C03652=1137.389,195.650,-63.085,-178.221,7.484,148.898
C03653=1137.385,195.899,-63.109,-178.219,7.486,148.898
C03654=1137.380,196.148,-63.132,-178.216,7.489,148.898
C03655=1137.375,196.397,-63.157,-178.213,7.491,148.898
C03656=1137.371,196.646,-63.181,-178.210,7.493,148.898
C03657=1137.366,196.895,-63.204,-178.207,7.496,148.897
C03658=1137.362,197.143,-63.229,-178.204,7.499,148.897
C03659=1137.357,197.392,-63.254,-178.202,7.501,148.897
C03660=1137.353,197.641,-63.278,-178.199,7.504,148.897
C03661=1137.348,197.890,-63.301,-178.196,7.506,148.896
C03662=1137.343,198.138,-63.325,-178.193,7.508,148.896
C03663=1137.338,198.387,-63.350,-178.191,7.511,148.896
C03664=1137.335,198.636,-63.374,-178.187,7.514,148.896
C03665=1137.330,198.885,-63.398,-178.184,7.517,148.896
C03666=1137.325,199.134,-63.422,-178.182,7.518,148.895
C03667=1137.320,199.382,-63.446,-178.179,7.521,148.895
C03668=1137.317,199.631,-63.471,-178.176,7.524,148.895
C03669=1137.311,199.880,-63.495,-178.173,7.526,148.895
C03670=1137.307,200.129,-63.519,-178.171,7.529,148.895
C03671=1137.303,200.377,-63.544,-178.167,7.531,148.894
C03672=1137.298,200.627,-63.568,-178.165,7.533,148.894
C03673=1137.293,200.875,-63.592,-178.162,7.536,148.894
C03674=1137.289,201.124,-63.616,-178.159,7.539,148.894
C03675=1137.284,201.373,-63.641,-178.156,7.542,148.894
C03676=1137.280,201.622,-63.665,-178.154,7.544,148.894
C03677=1137.275,201.870,-63.690,-178.151,7.546,148.893
C03678=1137.271,202.119,-63.714,-178.148,7.549,148.893
C03679=1137.267,202.368,-63.738,-178.145,7.551,148.893
C03680=1137.262,202.617,-63.763,-178.142,7.554,148.893
C03681=1137.257,202.865,-63.787,-178.140,7.557,148.893
C03682=1137.253,203.115,-63.812,-178.136,7.559,148.892
C03683=1137.248,203.363,-63.836,-178.134,7.561,148.892
C03684=1137.243,203.612,-63.861,-178.131,7.564,148.892
C03685=1137.239,203.861,-63.885,-178.128,7.567,148.892
C03686=1137.234,204.110,-63.910,-178.125,7.570,148.892
C03687=1137.230,204.358,-63.934,-178.123,7.572,148.891
C03688=1137.226,204.607,-63.960,-178.120,7.574,148.891
C03689=1137.221,204.855,-63.984,-178.117,7.577,148.891
C03690=1137.216,205.104,-64.009,-178.114,7.580,148.891
C03691=1137.212,205.353,-64.033,-178.111,7.582,148.891
C03692=1137.207,205.602,-64.058,-178.109,7.585,148.890
C03693=1137.203,205.850,-64.082,-178.106,7.588,148.890
C03694=1137.198,206.100,-64.107,-178.102,7.590,148.890
C03695=1137.194,206.347,-64.132,-178.100,7.592,148.890
C03696=1137.189,206.596,-64.156,-178.097,7.595,148.890
C03697=1137.185,206.845,-64.181,-178.094,7.598,148.890
C03698=1137.180,207.094,-64.205,-178.091,7.601,148.889
C03699=1137.176,207.343,-64.230,-178.089,7.603,148.889
C03700=1137.171,207.591,-64.255,-178.086,7.605,148.889
C03701=1137.166,207.840,-64.280,-178.083,7.608,148.889
C03702=1137.162,208.089,-64.305,-178.080,7.611,148.889
C03703=1137.158,208.337,-64.330,-178.078,7.613,148.889
C03704=1137.153,208.586,-64.355,-178.075,7.616,148.888
C03705=1137.148,208.835,-64.379,-178.072,7.619,148.888
C03706=1137.144,209.106,-64.406,-178.069,7.622,148.888
C03707=1137.138,209.376,-64.433,-178.066,7.624,148.888
C03708=1137.134,209.647,-64.460,-178.063,7.627,148.888
C03709=1137.129,209.918,-64.487,-178.060,7.630,148.887
C03710=1137.124,210.166,-64.513,-178.057,7.632,148.887
C03711=1137.120,210.416,-64.538,-178.054,7.635,148.887
C03712=1137.115,210.664,-64.563,-178.051,7.638,148.887
C03713=1137.111,210.912,-64.587,-178.048,7.641,148.887
C03714=1137.106,211.161,-64.612,-178.046,7.643,148.887
C03715=1137.101,211.410,-64.638,-178.043,7.646,148.886
C03716=1137.097,211.659,-64.663,-178.040,7.649,148.886
C03717=1137.093,211.907,-64.687,-178.037,7.651,148.886
C03718=1137.088,212.156,-64.712,-178.034,7.654,148.886
C03719=1137.083,212.404,-64.738,-178.032,7.656,148.886
C03720=1137.079,212.654,-64.763,-178.029,7.659,148.886
C03721=1137.075,212.902,-64.788,-178.026,7.662,148.885
C03722=1137.070,213.151,-64.813,-178.023,7.665,148.885
C03723=1137.066,213.400,-64.838,-178.020,7.668,148.885
C03724=1137.061,213.648,-64.864,-178.017,7.670,148.885
C03725=1137.057,213.897,-64.889,-178.015,7.672,148.885
C03726=1137.052,214.145,-64.914,-178.012,7.675,148.885
C03727=1137.048,214.394,-64.939,-178.009,7.678,148.885
C03728=1137.043,214.643,-64.964,-178.006,7.681,148.884
C03729=1137.039,214.891,-64.990,-178.003,7.683,148.884
C03730=1137.034,215.141,-65.015,-178.001,7.686,148.884
C03731=1137.030,215.389,-65.040,-177.998,7.688,148.884
C03732=1137.025,215.638,-65.066,-177.995,7.691,148.884
C03733=1137.020,215.886,-65.091,-177.992,7.694,148.884
C03734=1137.017,216.135,-65.116,-177.989,7.697,148.883
C03735=1137.012,216.383,-65.141,-177.986,7.700,148.883
C03736=1137.008,216.632,-65.167,-177.984,7.702,148.883
C03737=1137.003,216.881,-65.192,-177.981,7.705,148.883
C03738=1136.998,217.129,-65.217,-177.978,7.707,148.883
C03739=1136.994,217.378,-65.243,-177.975,7.710,148.883
C03740=1136.990,217.627,-65.269,-177.972,7.713,148.883
C03741=1136.985,217.876,-65.294,-177.969,7.716,148.882
C03742=1136.981,218.125,-65.319,-177.967,7.719,148.882
C03743=1136.976,218.373,-65.345,-177.964,7.721,148.882
C03744=1136.971,218.621,-65.370,-177.961,7.723,148.882
C03745=1136.967,218.870,-65.396,-177.958,7.726,148.882
C03746=1136.963,219.119,-65.422,-177.956,7.729,148.882
C03747=1136.958,219.367,-65.447,-177.953,7.732,148.882
C03748=1136.954,219.617,-65.472,-177.950,7.735,148.882
C03749=1136.949,219.865,-65.498,-177.947,7.738,148.881
C03750=1136.945,220.113,-65.523,-177.944,7.740,148.881
C03751=1136.940,220.362,-65.549,-177.942,7.743,148.881
C03752=1136.936,220.611,-65.575,-177.939,7.746,148.881
C03753=1136.931,220.859,-65.600,-177.936,7.748,148.881
C03754=1136.927,221.108,-65.626,-177.933,7.751,148.881
C03755=1136.923,221.357,-65.652,-177.930,7.754,148.880
C03756=1136.917,221.605,-65.678,-177.927,7.757,148.880
C03757=1136.913,221.854,-65.704,-177.924,7.760,148.880
C03758=1136.909,222.103,-65.729,-177.922,7.762,148.880
C03759=1136.905,222.352,-65.755,-177.919,7.765,148.880
C03760=1136.900,222.600,-65.780,-177.917,7.768,148.880
C03761=1136.896,222.849,-65.806,-177.913,7.770,148.880
C03762=1136.891,223.097,-65.832,-177.910,7.773,148.880
C03763=1136.887,223.346,-65.858,-177.908,7.776,148.879
C03764=1136.882,223.594,-65.884,-177.905,7.779,148.879
C03765=1136.878,223.843,-65.910,-177.902,7.782,148.879
C03766=1136.873,224.092,-65.936,-177.900,7.784,148.879
C03767=1136.869,224.340,-65.962,-177.897,7.787,148.879
C03768=1136.864,224.588,-65.987,-177.894,7.790,148.879
C03769=1136.859,224.838,-66.013,-177.891,7.792,148.879
C03770=1136.855,225.086,-66.039,-177.888,7.795,148.879
C03771=1136.851,225.335,-66.066,-177.885,7.798,148.878
C03772=1136.847,225.583,-66.091,-177.882,7.801,148.878
C03773=1136.842,225.832,-66.117,-177.880,7.804,148.878
C03774=1136.837,226.081,-66.143,-177.877,7.807,148.878
C03775=1136.833,226.329,-66.170,-177.874,7.810,148.878
C03776=1136.829,226.578,-66.195,-177.871,7.813,148.878
C03777=1136.824,226.827,-66.222,-177.869,7.815,148.878
C03778=1136.820,227.076,-66.247,-177.866,7.817,148.878
C03779=1136.815,227.323,-66.274,-177.863,7.820,148.877
C03780=1136.810,227.572,-66.300,-177.860,7.823,148.877
C03781=1136.806,227.821,-66.326,-177.857,7.826,148.877
C03782=1136.802,228.069,-66.352,-177.855,7.829,148.877
C03783=1136.798,228.318,-66.378,-177.852,7.832,148.877
C03784=1136.793,228.567,-66.404,-177.849,7.835,148.877
C03785=1136.789,228.815,-66.431,-177.846,7.838,148.877
C03786=1136.784,229.064,-66.457,-177.843,7.840,148.877
C03787=1136.780,229.312,-66.483,-177.841,7.843,148.877
C03788=1136.776,229.561,-66.509,-177.838,7.846,148.877
C03789=1136.771,229.809,-66.536,-177.835,7.849,148.877
C03790=1136.767,230.058,-66.562,-177.832,7.851,148.876
C03791=1136.762,230.307,-66.587,-177.829,7.854,148.876
C03792=1136.758,230.555,-66.614,-177.827,7.857,148.876
C03793=1136.754,230.804,-66.640,-177.824,7.860,148.876
C03794=1136.749,231.052,-66.667,-177.821,7.863,148.876
C03795=1136.745,231.301,-66.694,-177.818,7.865,148.876
C03796=1136.740,231.550,-66.720,-177.815,7.868,148.876
C03797=1136.736,231.798,-66.747,-177.813,7.871,148.876
C03798=1136.731,232.046,-66.773,-177.810,7.874,148.876
C03799=1136.727,232.295,-66.799,-177.807,7.877,148.875
C03800=1136.722,232.544,-66.825,-177.804,7.880,148.875
C03801=1136.718,232.792,-66.852,-177.801,7.883,148.875
C03802=1136.713,233.040,-66.879,-177.799,7.886,148.875
C03803=1136.709,233.289,-66.905,-177.796,7.889,148.875
C03804=1136.704,233.538,-66.932,-177.793,7.892,148.875
C03805=1136.700,233.786,-66.957,-177.790,7.895,148.875
C03806=1136.695,234.035,-66.985,-177.787,7.897,148.875
C03807=1136.691,234.283,-67.011,-177.785,7.900,148.875
C03808=1136.687,234.532,-67.038,-177.782,7.903,148.875
C03809=1136.682,234.780,-67.064,-177.779,7.906,148.875
C03810=1136.678,235.053,-67.094,-177.776,7.909,148.874
C03811=1136.673,235.324,-67.123,-177.773,7.912,148.874
C03812=1136.667,235.597,-67.151,-177.769,7.915,148.874
C03813=1136.664,235.869,-67.181,-177.767,7.918,148.874
C03814=1136.659,236.117,-67.208,-177.764,7.921,148.874
C03815=1136.654,236.366,-67.235,-177.761,7.924,148.874
C03816=1136.650,236.614,-67.261,-177.758,7.927,148.874
C03817=1136.645,236.863,-67.288,-177.755,7.930,148.874
C03818=1136.641,237.111,-67.315,-177.753,7.933,148.874
C03819=1136.637,237.360,-67.341,-177.750,7.936,148.874
C03820=1136.632,237.608,-67.368,-177.747,7.939,148.874
C03821=1136.628,237.857,-67.395,-177.744,7.942,148.873
C03822=1136.624,238.105,-67.422,-177.741,7.944,148.873
C03823=1136.619,238.353,-67.449,-177.739,7.947,148.873
C03824=1136.614,238.602,-67.476,-177.736,7.950,148.873
C03825=1136.610,238.851,-67.502,-177.733,7.953,148.873
C03826=1136.606,239.100,-67.529,-177.730,7.956,148.873
C03827=1136.601,239.348,-67.556,-177.727,7.959,148.873
C03828=1136.597,239.597,-67.583,-177.725,7.962,148.873
C03829=1136.593,239.845,-67.610,-177.722,7.965,148.873
C03830=1136.588,240.093,-67.637,-177.719,7.968,148.873
C03831=1136.583,240.342,-67.664,-177.716,7.971,148.873
C03832=1136.579,240.590,-67.691,-177.713,7.974,148.873
C03833=1136.575,240.839,-67.717,-177.711,7.976,148.872
C03834=1136.571,241.088,-67.745,-177.708,7.979,148.872
C03835=1136.567,241.336,-67.772,-177.705,7.982,148.872
C03836=1136.562,241.584,-67.799,-177.702,7.985,148.872
C03837=1136.557,241.833,-67.827,-177.699,7.988,148.872
C03838=1136.553,242.081,-67.853,-177.697,7.991,148.872
C03839=1136.549,242.329,-67.880,-177.694,7.994,148.872
C03840=1136.545,242.578,-67.907,-177.691,7.997,148.872
C03841=1136.540,242.827,-67.935,-177.689,8.000,148.872
C03842=1136.535,243.075,-67.962,-177.686,8.003,148.872
C03843=1136.531,243.323,-67.989,-177.683,8.006,148.872
C03844=1136.527,243.572,-68.016,-177.680,8.009,148.872
C03845=1136.523,243.821,-68.043,-177.677,8.012,148.872
C03846=1136.518,244.069,-68.070,-177.675,8.015,148.872
C03847=1136.514,244.317,-68.098,-177.672,8.018,148.872
C03848=1136.509,244.566,-68.125,-177.669,8.020,148.871
C03849=1136.505,244.814,-68.152,-177.666,8.023,148.871
C03850=1136.501,245.063,-68.180,-177.663,8.026,148.871
C03851=1136.496,245.311,-68.207,-177.661,8.029,148.871
C03852=1136.492,245.560,-68.235,-177.658,8.032,148.871
C03853=1136.487,245.808,-68.262,-177.654,8.036,148.871
C03854=1136.483,246.057,-68.290,-177.652,8.039,148.871
C03855=1136.478,246.305,-68.317,-177.649,8.042,148.871
C03856=1136.474,246.554,-68.344,-177.646,8.045,148.871
C03857=1136.470,246.802,-68.372,-177.644,8.048,148.871
C03858=1136.465,247.051,-68.399,-177.641,8.051,148.871
C03859=1136.461,247.299,-68.426,-177.638,8.054,148.871
C03860=1136.456,247.547,-68.454,-177.635,8.057,148.871
C03861=1136.452,247.796,-68.481,-177.632,8.059,148.871
C03862=1136.448,248.044,-68.509,-177.630,8.062,148.871
C03863=1136.443,248.293,-68.536,-177.627,8.065,148.871
C03864=1136.440,248.541,-68.564,-177.624,8.068,148.871
C03865=1136.435,248.790,-68.591,-177.622,8.071,148.871
C03866=1136.431,249.038,-68.619,-177.619,8.074,148.871
C03867=1136.427,249.287,-68.647,-177.616,8.077,148.870
C03868=1136.422,249.535,-68.674,-177.613,8.080,148.870
C03869=1136.418,249.783,-68.701,-177.611,8.083,148.870
C03870=1136.414,250.032,-68.730,-177.607,8.087,148.870
C03871=1136.408,250.281,-68.757,-177.604,8.090,148.870
C03872=1136.404,250.529,-68.785,-177.602,8.093,148.870
C03873=1136.400,250.778,-68.812,-177.599,8.096,148.870
C03874=1136.396,251.026,-68.840,-177.596,8.099,148.870
C03875=1136.391,251.273,-68.868,-177.594,8.102,148.870
C03876=1136.387,251.523,-68.895,-177.591,8.105,148.870
C03877=1136.383,251.771,-68.923,-177.588,8.108,148.870
C03878=1136.378,252.019,-68.952,-177.585,8.110,148.870
C03879=1136.374,252.268,-68.979,-177.582,8.113,148.870
C03880=1136.369,252.516,-69.007,-177.580,8.116,148.870
C03881=1136.366,252.764,-69.035,-177.577,8.120,148.870
C03882=1136.361,253.013,-69.062,-177.574,8.123,148.870
C03883=1136.356,253.262,-69.091,-177.571,8.126,148.870
C03884=1136.352,253.510,-69.118,-177.568,8.129,148.870
C03885=1136.348,253.758,-69.146,-177.565,8.132,148.870
C03886=1136.344,254.007,-69.174,-177.563,8.135,148.870
C03887=1136.339,254.255,-69.202,-177.560,8.138,148.870
C03888=1136.335,254.503,-69.230,-177.557,8.141,148.870
C03889=1136.331,254.751,-69.258,-177.555,8.144,148.870
C03890=1136.327,255.000,-69.286,-177.552,8.147,148.870
C03891=1136.322,255.248,-69.314,-177.549,8.150,148.869
C03892=1136.318,255.497,-69.342,-177.546,8.154,148.869
C03893=1136.313,255.745,-69.370,-177.543,8.157,148.870
C03894=1136.309,255.994,-69.398,-177.541,8.160,148.870
C03895=1136.304,256.242,-69.426,-177.538,8.163,148.869
C03896=1136.301,256.491,-69.454,-177.535,8.166,148.869
C03897=1136.296,256.739,-69.483,-177.532,8.168,148.869
C03898=1136.292,256.987,-69.511,-177.530,8.172,148.869
C03899=1136.287,257.235,-69.539,-177.527,8.175,148.869
C03900=1136.283,257.484,-69.567,-177.524,8.178,148.869
C03901=1136.279,257.732,-69.595,-177.521,8.181,148.869
C03902=1136.274,257.981,-69.624,-177.518,8.184,148.869
C03903=1136.270,258.229,-69.652,-177.515,8.187,148.869
C03904=1136.266,258.477,-69.680,-177.513,8.190,148.869
C03905=1136.261,258.725,-69.708,-177.510,8.193,148.869
C03906=1136.257,258.974,-69.736,-177.507,8.196,148.869
C03907=1136.252,259.222,-69.765,-177.504,8.199,148.869
C03908=1136.248,259.471,-69.793,-177.502,8.203,148.869
C03909=1136.243,259.719,-69.821,-177.499,8.206,148.869
C03910=1136.240,259.968,-69.849,-177.496,8.209,148.869
C03911=1136.235,260.216,-69.878,-177.493,8.212,148.869
C03912=1136.231,260.464,-69.906,-177.490,8.215,148.869
C03913=1136.227,260.713,-69.935,-177.488,8.218,148.869
C03914=1136.222,260.986,-69.966,-177.485,8.222,148.869
C03915=1136.216,261.260,-69.997,-177.482,8.225,148.869
C03916=1136.212,261.534,-70.028,-177.478,8.228,148.869
C03917=1136.207,261.807,-70.060,-177.475,8.232,148.869
C03918=1136.204,262.055,-70.088,-177.473,8.235,148.869
C03919=1136.199,262.304,-70.117,-177.470,8.238,148.869
C03920=1136.195,262.552,-70.145,-177.467,8.241,148.869
C03921=1136.191,262.800,-70.174,-177.464,8.244,148.869
C03922=1136.185,263.048,-70.203,-177.462,8.247,148.869
C03923=1136.182,263.297,-70.231,-177.459,8.251,148.869
C03924=1136.178,263.545,-70.260,-177.456,8.254,148.869
C03925=1136.173,263.793,-70.288,-177.453,8.257,148.869
C03926=1136.169,264.042,-70.317,-177.451,8.260,148.869
C03927=1136.165,264.290,-70.346,-177.448,8.263,148.869
C03928=1136.160,264.538,-70.374,-177.445,8.266,148.869
C03929=1136.156,264.787,-70.403,-177.442,8.270,148.869
C03930=1136.151,265.035,-70.432,-177.439,8.273,148.869
C03931=1136.147,265.283,-70.460,-177.437,8.276,148.869
C03932=1136.143,265.531,-70.490,-177.434,8.279,148.869
C03933=1136.138,265.780,-70.518,-177.431,8.282,148.869
C03934=1136.134,266.028,-70.546,-177.429,8.285,148.869
C03935=1136.130,266.277,-70.575,-177.425,8.289,148.869
C03936=1136.125,266.525,-70.604,-177.422,8.292,148.869
C03937=1136.121,266.774,-70.634,-177.420,8.295,148.869
C03938=1136.117,267.022,-70.661,-177.417,8.298,148.869
C03939=1136.113,267.270,-70.691,-177.414,8.301,148.869
C03940=1136.108,267.519,-70.720,-177.412,8.305,148.869
C03941=1136.103,267.766,-70.749,-177.409,8.308,148.869
C03942=1136.100,268.015,-70.777,-177.406,8.311,148.869
C03943=1136.096,268.263,-70.806,-177.404,8.314,148.869
C03944=1136.091,268.511,-70.836,-177.401,8.317,148.869
C03945=1136.086,268.760,-70.864,-177.397,8.321,148.869
C03946=1136.083,269.008,-70.893,-177.395,8.324,148.869
C03947=1136.079,269.256,-70.922,-177.392,8.327,148.869
C03948=1136.074,269.505,-70.951,-177.389,8.330,148.869
C03949=1136.070,269.753,-70.981,-177.387,8.333,148.869
C03950=1136.065,270.001,-71.009,-177.384,8.337,148.869
C03951=1136.061,270.249,-71.038,-177.381,8.340,148.869
C03952=1136.057,270.497,-71.067,-177.378,8.342,148.869
C03953=1136.053,270.746,-71.097,-177.376,8.346,148.869
C03954=1136.049,270.995,-71.126,-177.373,8.349,148.869
C03955=1136.044,271.242,-71.155,-177.370,8.353,148.869
C03956=1136.040,271.490,-71.184,-177.367,8.356,148.869
C03957=1136.035,271.739,-71.214,-177.365,8.359,148.869
C03958=1136.031,271.987,-71.242,-177.362,8.362,148.869
C03959=1136.027,272.236,-71.272,-177.359,8.365,148.869
C03960=1136.023,272.484,-71.301,-177.356,8.368,148.869
C03961=1136.019,272.731,-71.330,-177.354,8.372,148.870
C03962=1136.014,272.980,-71.359,-177.351,8.375,148.870
C03963=1136.010,273.228,-71.389,-177.348,8.378,148.869
C03964=1136.006,273.477,-71.417,-177.345,8.382,148.870
C03965=1136.002,273.725,-71.447,-177.342,8.385,148.870
C03966=1135.997,273.973,-71.476,-177.340,8.388,148.870
C03967=1135.993,274.222,-71.506,-177.337,8.391,148.870
C03968=1135.989,274.470,-71.535,-177.334,8.394,148.870
C03969=1135.985,274.718,-71.565,-177.331,8.398,148.870
C03970=1135.980,274.966,-71.594,-177.329,8.401,148.870
C03971=1135.976,275.214,-71.623,-177.326,8.404,148.870
C03972=1135.972,275.462,-71.653,-177.323,8.408,148.870
C03973=1135.967,275.710,-71.682,-177.320,8.410,148.870
C03974=1135.963,275.959,-71.711,-177.318,8.414,148.870
C03975=1135.959,276.207,-71.741,-177.315,8.417,148.870
C03976=1135.954,276.456,-71.771,-177.312,8.421,148.870
C03977=1135.950,276.704,-71.800,-177.309,8.424,148.870
C03978=1135.946,276.952,-71.830,-177.306,8.427,148.870
C03979=1135.942,277.200,-71.859,-177.304,8.430,148.870
C03980=1135.937,277.449,-71.889,-177.301,8.434,148.870
C03981=1135.934,277.696,-71.919,-177.298,8.437,148.870
C03982=1135.929,277.945,-71.948,-177.296,8.440,148.870
C03983=1135.925,278.193,-71.978,-177.293,8.443,148.870
C03984=1135.921,278.441,-72.007,-177.290,8.447,148.870
C03985=1135.917,278.689,-72.037,-177.287,8.450,148.870
C03986=1135.912,278.938,-72.067,-177.285,8.453,148.871
C03987=1135.908,279.186,-72.097,-177.282,8.456,148.870
C03988=1135.904,279.434,-72.126,-177.279,8.460,148.871
C03989=1135.900,279.682,-72.156,-177.276,8.463,148.871
C03990=1135.896,279.930,-72.185,-177.274,8.466,148.871
C03991=1135.891,280.179,-72.215,-177.270,8.470,148.871
C03992=1135.887,280.427,-72.246,-177.268,8.473,148.871
C03993=1135.883,280.675,-72.275,-177.265,8.476,148.871
C03994=1135.878,280.923,-72.304,-177.263,8.479,148.871
C03995=1135.874,281.171,-72.335,-177.260,8.483,148.871
C03996=1135.870,281.419,-72.365,-177.257,8.486,148.871
C03997=1135.865,281.668,-72.394,-177.254,8.489,148.871
C03998=1135.862,281.915,-72.424,-177.251,8.493,148.871
C03999=1135.857,282.164,-72.454,-177.249,8.496,148.871
C04000=1135.852,282.412,-72.484,-177.246,8.499,148.871
C04001=1135.849,282.660,-72.514,-177.244,8.502,148.871
C04002=1135.844,282.908,-72.544,-177.240,8.506,148.871
C04003=1135.840,283.156,-72.574,-177.238,8.509,148.872
C04004=1135.836,283.405,-72.604,-177.235,8.512,148.871
C04005=1135.832,283.653,-72.635,-177.232,8.516,148.872
C04006=1135.825,284.060,-72.683,-177.228,8.522,148.872
C04007=1135.804,285.282,-72.833,-178.121,10.280,149.550
C04008=1135.800,285.531,-72.864,-178.118,10.283,149.550
C04009=1135.796,285.779,-72.894,-178.115,10.285,149.550
C04010=1135.791,286.027,-72.925,-178.112,10.288,149.550
C04011=1135.786,286.275,-72.955,-178.109,10.290,149.550
C04012=1135.783,286.524,-72.986,-178.106,10.293,149.549
C04013=1135.779,286.772,-73.017,-178.103,10.296,149.549
C04014=1135.775,287.019,-73.047,-178.100,10.298,149.549
C04015=1135.771,287.268,-73.078,-178.096,10.301,149.549
C04016=1135.766,287.516,-73.109,-178.093,10.304,149.549
C04017=1135.762,287.763,-73.139,-178.091,10.305,149.548
C04018=1135.758,288.012,-73.170,-178.088,10.308,149.548
C04019=1135.754,288.260,-73.201,-178.084,10.310,149.548
C04020=1135.750,288.508,-73.231,-178.081,10.313,149.548
C04021=1135.746,288.756,-73.262,-178.078,10.316,149.548
C04022=1135.741,289.004,-73.293,-178.075,10.318,149.548
C04023=1135.736,289.252,-73.324,-178.072,10.321,149.547
C04024=1135.733,289.501,-73.354,-178.069,10.324,149.547
C04025=1135.729,289.748,-73.386,-178.066,10.326,149.547
C04026=1135.724,289.996,-73.416,-178.063,10.329,149.547
C04027=1135.720,290.245,-73.448,-178.060,10.331,149.547
C04028=1135.716,290.492,-73.478,-178.056,10.334,149.546
C04029=1135.712,290.740,-73.508,-178.054,10.336,149.546
C04030=1135.708,290.989,-73.540,-178.051,10.338,149.546
C04031=1135.703,291.236,-73.571,-178.048,10.341,149.546
C04032=1135.700,291.485,-73.602,-178.044,10.343,149.546
C04033=1135.696,291.732,-73.632,-178.041,10.346,149.546
C04034=1135.691,291.980,-73.663,-178.038,10.349,149.545
C04035=1135.687,292.229,-73.694,-178.035,10.351,149.545
C04036=1135.683,292.476,-73.726,-178.032,10.354,149.545
C04037=1135.679,292.725,-73.757,-178.029,10.357,149.545
C04038=1135.675,292.973,-73.787,-178.026,10.359,149.545
C04039=1135.671,293.221,-73.819,-178.023,10.362,149.544
C04040=1135.667,293.452,-73.847,-178.020,10.364,149.544
C04041=1135.663,293.683,-73.877,-178.017,10.366,149.544
C04042=1135.659,293.914,-73.905,-178.014,10.369,149.544
C04043=1135.656,294.145,-73.935,-178.012,10.371,149.544
C04044=1135.651,294.377,-73.964,-178.008,10.373,149.544
C04045=1135.647,294.607,-73.993,-178.005,10.376,149.544
C04046=1135.643,294.839,-74.021,-178.003,10.378,149.543
C04047=1135.639,295.070,-74.051,-178.000,10.381,149.543
C04048=1135.636,295.318,-74.083,-177.996,10.383,149.543
C04049=1135.631,295.566,-74.113,-177.994,10.386,149.543
C04050=1135.627,295.814,-74.144,-177.991,10.389,149.543
C04051=1135.623,296.062,-74.176,-177.987,10.391,149.542
C04052=1135.619,296.310,-74.207,-177.984,10.394,149.542
C04053=1135.614,296.558,-74.239,-177.981,10.396,149.542
C04054=1135.610,296.806,-74.270,-177.979,10.398,149.542
C04055=1135.606,297.054,-74.301,-177.975,10.401,149.542
C04056=1135.602,297.302,-74.332,-177.972,10.403,149.542
C04057=1135.598,297.550,-74.364,-177.969,10.406,149.541
C04058=1135.594,297.798,-74.396,-177.966,10.408,149.541
C04059=1135.590,298.046,-74.426,-177.963,10.411,149.541
C04060=1135.586,298.294,-74.458,-177.959,10.413,149.541
C04061=1135.581,298.542,-74.489,-177.957,10.416,149.541
C04062=1135.578,298.790,-74.521,-177.953,10.419,149.540
C04063=1135.573,299.037,-74.552,-177.950,10.421,149.540
C04064=1135.569,299.286,-74.583,-177.947,10.424,149.540
C04065=1135.565,299.533,-74.615,-177.944,10.427,149.540
C04066=1135.561,299.781,-74.647,-177.941,10.429,149.540
C04067=1135.557,300.030,-74.678,-177.938,10.432,149.540
C04068=1135.553,300.277,-74.709,-177.934,10.434,149.539
C04069=1135.549,300.525,-74.741,-177.931,10.437,149.539
C04070=1135.544,300.773,-74.773,-177.929,10.439,149.539
C04071=1135.540,301.021,-74.804,-177.926,10.441,149.539
C04072=1135.536,301.269,-74.836,-177.922,10.444,149.539
C04073=1135.532,301.517,-74.868,-177.920,10.447,149.538
C04074=1135.528,301.765,-74.900,-177.916,10.449,149.538
C04075=1135.524,302.013,-74.930,-177.913,10.452,149.538
C04076=1135.519,302.261,-74.963,-177.910,10.454,149.538
C04077=1135.516,302.509,-74.995,-177.907,10.457,149.538
C04078=1135.511,302.756,-75.026,-177.904,10.459,149.538
C04079=1135.508,303.004,-75.058,-177.900,10.462,149.537
C04080=1135.503,303.253,-75.090,-177.897,10.465,149.537
C04081=1135.499,303.501,-75.121,-177.894,10.467,149.537
C04082=1135.495,303.749,-75.153,-177.891,10.470,149.537
C04083=1135.491,303.997,-75.185,-177.888,10.472,149.537
C04084=1135.486,304.245,-75.217,-177.885,10.475,149.536
C04085=1135.482,304.493,-75.249,-177.882,10.477,149.536
C04086=1135.479,304.741,-75.281,-177.879,10.479,149.536
C04087=1135.474,304.988,-75.312,-177.876,10.482,149.536
C04088=1135.470,305.236,-75.345,-177.873,10.485,149.536
C04089=1135.466,305.484,-75.376,-177.870,10.487,149.536
C04090=1135.462,305.732,-75.408,-177.866,10.489,149.535
C04091=1135.457,305.980,-75.440,-177.863,10.492,149.535
C04092=1135.454,306.228,-75.472,-177.860,10.495,149.535
C04093=1135.449,306.475,-75.504,-177.857,10.497,149.535
C04094=1135.445,306.724,-75.536,-177.854,10.500,149.535
C04095=1135.441,306.972,-75.568,-177.851,10.503,149.534
C04096=1135.437,307.185,-75.596,-177.848,10.504,149.534
C04097=1135.434,307.398,-75.624,-177.845,10.507,149.534
C04098=1135.430,307.613,-75.651,-177.843,10.509,149.534
C04099=1135.427,307.826,-75.679,-177.840,10.511,149.534
C04100=1135.423,308.039,-75.707,-177.837,10.513,149.534
C04101=1135.420,308.253,-75.734,-177.835,10.515,149.534
C04102=1135.416,308.467,-75.762,-177.832,10.518,149.533
C04103=1135.414,308.681,-75.790,-177.829,10.520,149.533
C04104=1135.409,308.928,-75.822,-177.826,10.522,149.533
C04105=1135.405,309.176,-75.854,-177.823,10.525,149.533
C04106=1135.400,309.425,-75.886,-177.820,10.527,149.533
C04107=1135.397,309.673,-75.918,-177.816,10.530,149.532
C04108=1135.392,309.920,-75.951,-177.814,10.533,149.532
C04109=1135.388,310.168,-75.983,-177.810,10.535,149.532
C04110=1135.384,310.416,-76.015,-177.807,10.538,149.532
C04111=1135.380,310.663,-76.048,-177.804,10.540,149.532
C04112=1135.376,310.912,-76.080,-177.801,10.543,149.532
C04113=1135.372,311.160,-76.112,-177.798,10.546,149.531
C04114=1135.368,311.407,-76.145,-177.794,10.548,149.531
C04115=1135.364,311.655,-76.177,-177.791,10.551,149.531
C04116=1135.359,311.903,-76.209,-177.788,10.553,149.531
C04117=1135.356,312.151,-76.242,-177.785,10.556,149.531
C04118=1135.352,312.399,-76.274,-177.782,10.558,149.530
C04119=1135.348,312.646,-76.307,-177.779,10.560,149.530
C04120=1135.343,312.894,-76.339,-177.776,10.563,149.530
C04121=1135.339,313.142,-76.371,-177.773,10.565,149.530
C04122=1135.335,313.390,-76.404,-177.770,10.568,149.530
C04123=1135.331,313.638,-76.436,-177.767,10.570,149.529
C04124=1135.327,313.886,-76.469,-177.763,10.573,149.529
C04125=1135.323,314.134,-76.501,-177.760,10.576,149.529
C04126=1135.320,314.381,-76.534,-177.757,10.578,149.529
C04127=1135.315,314.630,-76.566,-177.754,10.581,149.529
C04128=1135.311,314.878,-76.599,-177.751,10.583,149.528
C04129=1135.307,315.126,-76.631,-177.747,10.586,149.528
C04130=1135.303,315.373,-76.664,-177.744,10.589,149.528
C04131=1135.298,315.620,-76.697,-177.741,10.591,149.528
C04132=1135.295,315.868,-76.729,-177.738,10.593,149.528
C04133=1135.291,316.116,-76.762,-177.735,10.596,149.528
C04134=1135.286,316.364,-76.794,-177.732,10.599,149.527
C04135=1135.283,316.612,-76.827,-177.729,10.601,149.527
C04136=1135.279,316.860,-76.860,-177.725,10.604,149.527
C04137=1135.274,317.108,-76.893,-177.722,10.606,149.527
C04138=1135.271,317.355,-76.925,-177.719,10.609,149.527
C04139=1135.267,317.603,-76.958,-177.716,10.611,149.526
C04140=1135.262,317.851,-76.992,-177.712,10.614,149.526
C04141=1135.258,318.099,-77.024,-177.710,10.616,149.526
C04142=1135.255,318.347,-77.057,-177.707,10.618,149.526
C04143=1135.250,318.594,-77.090,-177.703,10.621,149.526
C04144=1135.246,318.842,-77.123,-177.701,10.624,149.525
C04145=1135.242,319.090,-77.155,-177.697,10.626,149.525
C04146=1135.238,319.338,-77.188,-177.694,10.628,149.525
C04147=1135.234,319.586,-77.221,-177.691,10.631,149.525
C04148=1135.230,319.833,-77.254,-177.688,10.634,149.525
C04149=1135.226,320.081,-77.287,-177.684,10.636,149.524
C04150=1135.222,320.329,-77.320,-177.681,10.639,149.524
C04151=1135.217,320.577,-77.353,-177.678,10.641,149.524
C04152=1135.214,320.790,-77.382,-177.676,10.643,149.524
C04153=1135.211,321.004,-77.410,-177.672,10.646,149.524
C04154=1135.208,321.217,-77.438,-177.670,10.648,149.524
C04155=1135.204,321.430,-77.467,-177.667,10.650,149.523
C04156=1135.201,321.644,-77.495,-177.665,10.652,149.523
C04157=1135.197,321.858,-77.523,-177.662,10.655,149.523
C04158=1135.194,322.071,-77.552,-177.659,10.657,149.523
C04159=1135.190,322.285,-77.581,-177.657,10.659,149.523
C04160=1135.186,322.533,-77.614,-177.653,10.661,149.523
C04161=1135.182,322.781,-77.647,-177.650,10.663,149.522
C04162=1135.178,323.028,-77.680,-177.647,10.666,149.522
C04163=1135.174,323.276,-77.714,-177.644,10.669,149.522
C04164=1135.170,323.523,-77.746,-177.640,10.671,149.522
C04165=1135.166,323.771,-77.779,-177.637,10.674,149.522
C04166=1135.162,324.019,-77.812,-177.634,10.676,149.521
C04167=1135.158,324.266,-77.846,-177.631,10.679,149.521
C04168=1135.155,324.514,-77.880,-177.628,10.682,149.521
C04169=1135.151,324.762,-77.913,-177.625,10.684,149.521
C04170=1135.146,325.010,-77.946,-177.621,10.686,149.521
C04171=1135.142,325.258,-77.979,-177.618,10.689,149.520
C04172=1135.138,325.505,-78.012,-177.615,10.692,149.520
C04173=1135.134,325.753,-78.046,-177.612,10.694,149.520
C04174=1135.130,326.000,-78.079,-177.608,10.697,149.520
C04175=1135.127,326.249,-78.113,-177.605,10.699,149.520
C04176=1135.123,326.496,-78.146,-177.602,10.702,149.520
C04177=1135.118,326.744,-78.180,-177.599,10.704,149.519
C04178=1135.113,326.992,-78.213,-177.596,10.707,149.519
C04179=1135.110,327.239,-78.247,-177.593,10.709,149.519
C04180=1135.106,327.487,-78.280,-177.589,10.712,149.519
C04181=1135.102,327.735,-78.314,-177.586,10.714,149.518
C04182=1135.098,327.982,-78.347,-177.583,10.717,149.518
C04183=1135.094,328.230,-78.381,-177.580,10.720,149.518
C04184=1135.090,328.478,-78.414,-177.576,10.722,149.518
C04185=1135.086,328.725,-78.448,-177.573,10.725,149.518
C04186=1135.082,328.974,-78.482,-177.570,10.727,149.518
C04187=1135.078,329.221,-78.515,-177.567,10.729,149.517
C04188=1135.074,329.469,-78.549,-177.564,10.731,149.517
C04189=1135.070,329.716,-78.582,-177.561,10.734,149.517
C04190=1135.066,329.965,-78.615,-177.558,10.737,149.517
C04191=1135.062,330.212,-78.649,-177.554,10.739,149.517
C04192=1135.057,330.460,-78.683,-177.551,10.741,149.516
C04193=1135.054,330.707,-78.717,-177.548,10.744,149.516
C04194=1135.050,330.955,-78.750,-177.545,10.747,149.516
C04195=1135.046,331.203,-78.784,-177.542,10.749,149.516
C04196=1135.041,331.451,-78.818,-177.538,10.752,149.516
C04197=1135.038,331.698,-78.852,-177.535,10.754,149.515
C04198=1135.034,331.946,-78.885,-177.532,10.757,149.515
C04199=1135.030,332.193,-78.919,-177.529,10.759,149.515
C04200=1135.025,332.441,-78.953,-177.525,10.762,149.515
C04201=1135.021,332.688,-78.987,-177.522,10.765,149.515
C04202=1135.018,332.936,-79.021,-177.519,10.767,149.514
C04203=1135.014,333.184,-79.054,-177.516,10.769,149.514
C04204=1135.009,333.431,-79.089,-177.512,10.772,149.514
C04205=1135.006,333.680,-79.122,-177.510,10.775,149.514
C04206=1135.002,333.927,-79.156,-177.506,10.777,149.514
C04207=1134.998,334.174,-79.191,-177.503,10.780,149.513
C04208=1134.995,334.388,-79.220,-177.501,10.782,149.513
C04209=1134.991,334.601,-79.249,-177.497,10.784,149.513
C04210=1134.987,334.815,-79.279,-177.495,10.786,149.513
C04211=1134.985,335.028,-79.308,-177.492,10.788,149.513
C04212=1134.981,335.241,-79.337,-177.489,10.790,149.513
C04213=1134.977,335.455,-79.367,-177.486,10.793,149.512
C04214=1134.974,335.668,-79.396,-177.483,10.795,149.512
C04215=1134.971,335.882,-79.425,-177.481,10.797,149.512
C04216=1134.966,336.129,-79.459,-177.478,10.799,149.512
C04217=1134.963,336.376,-79.493,-177.474,10.801,149.512
C04218=1134.959,336.624,-79.527,-177.472,10.804,149.512
C04219=1134.954,336.872,-79.561,-177.468,10.807,149.511
C04220=1134.951,337.120,-79.595,-177.465,10.809,149.511
C04221=1134.947,337.367,-79.630,-177.462,10.812,149.511
C04222=1134.943,337.614,-79.664,-177.458,10.814,149.511
C04223=1134.939,337.862,-79.699,-177.455,10.817,149.511
C04224=1134.935,338.109,-79.732,-177.452,10.819,149.510
C04225=1134.931,338.358,-79.767,-177.449,10.822,149.510
C04226=1134.927,338.605,-79.801,-177.445,10.824,149.510
C04227=1134.923,338.853,-79.835,-177.442,10.827,149.510
C04228=1134.919,339.101,-79.869,-177.439,10.829,149.510
C04229=1134.914,339.348,-79.904,-177.436,10.832,149.509
C04230=1134.911,339.596,-79.938,-177.433,10.834,149.509
C04231=1134.907,339.843,-79.972,-177.429,10.837,149.509
C04232=1134.903,340.091,-80.006,-177.426,10.839,149.509
C04233=1134.899,340.338,-80.041,-177.423,10.842,149.508
C04234=1134.895,340.587,-80.076,-177.420,10.844,149.508
C04235=1134.891,340.834,-80.110,-177.416,10.847,149.508
C04236=1134.887,341.081,-80.145,-177.413,10.849,149.508
C04237=1134.884,341.328,-80.179,-177.410,10.852,149.508
C04238=1134.880,341.576,-80.214,-177.406,10.854,149.507
C04239=1134.875,341.824,-80.248,-177.403,10.857,149.507
C04240=1134.872,342.072,-80.283,-177.400,10.860,149.507
C04241=1134.867,342.319,-80.317,-177.397,10.862,149.507
C04242=1134.863,342.567,-80.352,-177.394,10.864,149.507
C04243=1134.859,342.814,-80.386,-177.390,10.867,149.506
C04244=1134.856,343.062,-80.421,-177.387,10.869,149.506
C04245=1134.851,343.309,-80.456,-177.384,10.872,149.506
C04246=1134.848,343.557,-80.490,-177.381,10.875,149.506
C04247=1134.843,343.804,-80.524,-177.377,10.877,149.506
C04248=1134.839,344.053,-80.559,-177.374,10.880,149.505
C04249=1134.836,344.299,-80.594,-177.371,10.882,149.505
C04250=1134.832,344.547,-80.629,-177.367,10.884,149.505
C04251=1134.827,344.795,-80.663,-177.364,10.887,149.505
C04252=1134.824,345.042,-80.698,-177.361,10.889,149.504
C04253=1134.820,345.289,-80.733,-177.358,10.892,149.504
C04254=1134.816,345.537,-80.767,-177.355,10.895,149.504
C04255=1134.812,345.785,-80.803,-177.351,10.897,149.504
C04256=1134.808,346.032,-80.837,-177.348,10.899,149.504
C04257=1134.804,346.280,-80.872,-177.345,10.902,149.503
C04258=1134.800,346.527,-80.907,-177.341,10.904,149.503
C04259=1134.796,346.775,-80.942,-177.339,10.906,149.503
C04260=1134.792,347.023,-80.977,-177.335,10.909,149.503
C04261=1134.789,347.270,-81.011,-177.332,10.911,149.503
C04262=1134.785,347.518,-81.046,-177.329,10.914,149.502
C04263=1134.780,347.764,-81.081,-177.326,10.916,149.502
C04264=1134.777,347.978,-81.112,-177.322,10.919,149.502
C04265=1134.773,348.192,-81.142,-177.320,10.921,149.502
C04266=1134.771,348.405,-81.172,-177.317,10.923,149.502
C04267=1134.767,348.617,-81.202,-177.314,10.925,149.501
C04268=1134.763,348.831,-81.232,-177.311,10.928,149.501
C04269=1134.760,349.044,-81.262,-177.309,10.929,149.501
C04270=1134.757,349.257,-81.292,-177.306,10.931,149.501
C04271=1134.754,349.471,-81.323,-177.303,10.934,149.501
C04272=1134.749,349.718,-81.357,-177.299,10.936,149.500
C04273=1134.746,349.966,-81.393,-177.295,10.939,149.500
C04274=1134.742,350.213,-81.428,-177.292,10.942,149.500
C04275=1134.737,350.460,-81.463,-177.288,10.945,149.500
C04276=1134.734,350.708,-81.498,-177.284,10.947,149.499
C04277=1134.730,350.955,-81.534,-177.280,10.950,149.499
C04278=1134.726,351.203,-81.568,-177.277,10.953,149.499
C04279=1134.722,351.450,-81.604,-177.273,10.956,149.499
C04280=1134.719,351.698,-81.639,-177.269,10.958,149.498
C04281=1134.715,351.946,-81.674,-177.266,10.961,149.498
C04282=1134.711,352.193,-81.709,-177.262,10.963,149.498
C04283=1134.707,352.440,-81.744,-177.258,10.967,149.498
C04284=1134.703,352.688,-81.780,-177.255,10.969,149.497
C04285=1134.699,352.936,-81.815,-177.251,10.971,149.497
C04286=1134.694,353.183,-81.850,-177.247,10.974,149.497
C04287=1134.691,353.430,-81.886,-177.244,10.977,149.497
C04288=1134.687,353.678,-81.922,-177.240,10.979,149.496
C04289=1134.683,353.925,-81.957,-177.236,10.982,149.496
C04290=1134.679,354.172,-81.992,-177.233,10.985,149.496
C04291=1134.676,354.420,-82.028,-177.229,10.987,149.495
C04292=1134.672,354.668,-82.063,-177.225,10.990,149.495
C04293=1134.668,354.915,-82.098,-177.222,10.993,149.495
C04294=1134.664,355.163,-82.134,-177.218,10.995,149.494
C04295=1134.660,355.409,-82.169,-177.215,10.997,149.494
C04296=1134.656,355.657,-82.205,-177.211,11.000,149.494
C04297=1134.653,355.904,-82.240,-177.207,11.003,149.494
C04298=1134.648,356.152,-82.276,-177.204,11.005,149.493
C04299=1134.645,356.400,-82.312,-177.200,11.008,149.493
C04300=1134.641,356.647,-82.347,-177.196,11.011,149.493
C04301=1134.637,356.894,-82.382,-177.193,11.013,149.493
C04302=1134.633,357.142,-82.418,-177.189,11.015,149.492
C04303=1134.629,357.389,-82.454,-177.186,11.018,149.492
C04304=1134.625,357.636,-82.490,-177.182,11.020,149.492
C04305=1134.622,357.884,-82.526,-177.179,11.023,149.492
C04306=1134.618,358.131,-82.562,-177.175,11.026,149.491
C04307=1134.614,358.379,-82.597,-177.171,11.028,149.491
C04308=1134.610,358.627,-82.633,-177.168,11.030,149.491
C04309=1134.606,358.873,-82.668,-177.165,11.033,149.491
C04310=1134.602,359.121,-82.704,-177.162,11.035,149.490
C04311=1134.599,359.368,-82.740,-177.158,11.037,149.490
C04312=1134.594,359.616,-82.776,-177.155,11.040,149.490
C04313=1134.591,359.863,-82.812,-177.151,11.042,149.489
C04314=1134.587,360.111,-82.847,-177.148,11.044,149.489
C04315=1134.583,360.357,-82.884,-177.144,11.048,149.489
C04316=1134.579,360.605,-82.920,-177.140,11.050,149.489
C04317=1134.575,360.853,-82.955,-177.137,11.053,149.488
C04318=1134.572,361.100,-82.992,-177.133,11.055,149.488
C04319=1134.568,361.347,-83.028,-177.130,11.057,149.488
C04320=1134.564,361.561,-83.058,-177.127,11.059,149.488
C04321=1134.561,361.773,-83.090,-177.124,11.061,149.487
C04322=1134.558,361.987,-83.120,-177.122,11.063,149.487
C04323=1134.555,362.199,-83.151,-177.119,11.065,149.487
C04324=1134.552,362.413,-83.182,-177.116,11.068,149.487
C04325=1134.548,362.626,-83.214,-177.113,11.069,149.487
C04326=1134.544,362.839,-83.244,-177.110,11.072,149.486
C04327=1134.541,363.052,-83.276,-177.107,11.073,149.486
C04328=1134.538,363.299,-83.311,-177.104,11.076,149.486
C04329=1134.534,363.546,-83.348,-177.100,11.078,149.486
C04330=1134.530,363.794,-83.384,-177.097,11.080,149.485
C04331=1134.527,364.041,-83.420,-177.093,11.083,149.485
C04332=1134.522,364.288,-83.456,-177.090,11.085,149.485
C04333=1134.519,364.535,-83.492,-177.087,11.088,149.485
C04334=1134.514,364.783,-83.529,-177.084,11.090,149.484
C04335=1134.511,365.030,-83.565,-177.081,11.092,149.484
C04336=1134.507,365.277,-83.602,-177.078,11.095,149.484
C04337=1134.503,365.525,-83.637,-177.074,11.097,149.484
C04338=1134.499,365.772,-83.674,-177.071,11.099,149.483
C04339=1134.496,366.019,-83.710,-177.067,11.102,149.483
C04340=1134.491,366.267,-83.746,-177.064,11.104,149.483
C04341=1134.489,366.514,-83.783,-177.061,11.106,149.483
C04342=1134.484,366.762,-83.819,-177.058,11.108,149.482
C04343=1134.481,367.009,-83.855,-177.055,11.111,149.482
C04344=1134.477,367.256,-83.892,-177.051,11.113,149.482
C04345=1134.473,367.503,-83.928,-177.048,11.116,149.482
C04346=1134.469,367.751,-83.965,-177.045,11.117,149.482
C04347=1134.465,367.998,-84.002,-177.042,11.120,149.481
C04348=1134.461,368.245,-84.037,-177.039,11.122,149.481
C04349=1134.457,368.493,-84.074,-177.036,11.125,149.481
C04350=1134.454,368.739,-84.110,-177.033,11.126,149.481
C04351=1134.450,368.987,-84.147,-177.030,11.129,149.480
C04352=1134.446,369.235,-84.184,-177.026,11.131,149.480
C04353=1134.443,369.482,-84.220,-177.024,11.133,149.480
C04354=1134.439,369.729,-84.257,-177.020,11.136,149.480
C04355=1134.434,369.976,-84.294,-177.017,11.138,149.480
C04356=1134.431,370.223,-84.330,-177.014,11.141,149.479
C04357=1134.427,370.470,-84.367,-177.011,11.142,149.479
C04358=1134.423,370.718,-84.403,-177.008,11.145,149.479
C04359=1134.420,370.966,-84.440,-177.005,11.148,149.479
C04360=1134.416,371.213,-84.476,-177.002,11.149,149.479
C04361=1134.412,371.460,-84.513,-176.999,11.152,149.478
C04362=1134.408,371.707,-84.549,-176.996,11.154,149.478
C04363=1134.404,371.954,-84.586,-176.993,11.156,149.478
C04364=1134.400,372.202,-84.623,-176.990,11.158,149.478
C04365=1134.397,372.449,-84.660,-176.987,11.160,149.478
C04366=1134.393,372.696,-84.697,-176.984,11.163,149.478
C04367=1134.389,372.943,-84.734,-176.981,11.165,149.477
C04368=1134.385,373.191,-84.770,-176.978,11.167,149.477
C04369=1134.382,373.438,-84.807,-176.975,11.170,149.477
C04370=1134.378,373.685,-84.844,-176.972,11.172,149.477
C04371=1134.374,373.933,-84.881,-176.969,11.174,149.477
C04372=1134.370,374.180,-84.918,-176.966,11.177,149.477
C04373=1134.367,374.427,-84.954,-176.964,11.179,149.476
C04374=1134.363,374.675,-84.991,-176.960,11.181,149.476
C04375=1134.359,374.922,-85.028,-176.958,11.183,149.476
C04376=1134.355,375.135,-85.060,-176.955,11.185,149.476
C04377=1134.353,375.347,-85.092,-176.953,11.187,149.476
C04378=1134.349,375.560,-85.124,-176.950,11.188,149.476
C04379=1134.346,375.773,-85.155,-176.948,11.190,149.475
C04380=1134.343,375.986,-85.187,-176.945,11.193,149.475
C04381=1134.339,376.199,-85.218,-176.943,11.195,149.475
C04382=1134.336,376.411,-85.251,-176.940,11.197,149.475
C04383=1134.334,376.624,-85.283,-176.938,11.199,149.475
C04384=1134.329,376.872,-85.320,-176.935,11.201,149.475
C04385=1134.325,377.119,-85.356,-176.932,11.204,149.475
C04386=1134.321,377.366,-85.393,-176.930,11.205,149.475
C04387=1134.318,377.613,-85.431,-176.927,11.208,149.475
C04388=1134.314,377.860,-85.468,-176.924,11.210,149.474
C04389=1134.310,378.108,-85.505,-176.922,11.212,149.474
C04390=1134.306,378.356,-85.542,-176.919,11.215,149.474
C04391=1134.303,378.602,-85.580,-176.916,11.216,149.474
C04392=1134.299,378.849,-85.616,-176.913,11.219,149.474
C04393=1134.295,379.096,-85.653,-176.911,11.221,149.474
C04394=1134.292,379.343,-85.691,-176.908,11.224,149.474
C04395=1134.288,379.591,-85.728,-176.906,11.226,149.474
C04396=1134.284,379.838,-85.765,-176.903,11.228,149.474
C04397=1134.281,380.085,-85.802,-176.900,11.230,149.473
C04398=1134.277,380.332,-85.839,-176.898,11.232,149.473
C04399=1134.273,380.579,-85.877,-176.895,11.235,149.473
C04400=1134.269,380.827,-85.914,-176.893,11.237,149.473
C04401=1134.265,381.074,-85.951,-176.889,11.239,149.473
C04402=1134.261,381.321,-85.989,-176.887,11.242,149.473
C04403=1134.258,381.568,-86.026,-176.885,11.244,149.473
C04404=1134.254,381.815,-86.063,-176.882,11.246,149.473
C04405=1134.251,382.063,-86.101,-176.880,11.248,149.473
C04406=1134.247,382.309,-86.138,-176.877,11.251,149.473
C04407=1134.243,382.557,-86.175,-176.874,11.253,149.473
C04408=1134.239,382.804,-86.213,-176.872,11.255,149.473
C04409=1134.235,383.051,-86.250,-176.869,11.258,149.473
C04410=1134.232,383.298,-86.287,-176.867,11.260,149.473
C04411=1134.228,383.546,-86.325,-176.865,11.261,149.473
C04412=1134.224,383.792,-86.363,-176.864,11.263,149.473
C04413=1134.220,384.040,-86.400,-176.863,11.265,149.473
C04414=1134.216,384.287,-86.438,-176.862,11.266,149.473
C04415=1134.212,384.534,-86.474,-176.861,11.268,149.473
C04416=1134.209,384.781,-86.512,-176.860,11.270,149.473
C04417=1134.205,385.029,-86.549,-176.859,11.271,149.473
C04418=1134.202,385.276,-86.587,-176.858,11.272,149.474
C04419=1134.198,385.522,-86.625,-176.857,11.274,149.474
C04420=1134.194,385.770,-86.662,-176.856,11.276,149.474
C04421=1134.191,386.017,-86.700,-176.855,11.278,149.474
C04422=1134.187,386.264,-86.736,-176.855,11.279,149.474
C04423=1134.183,386.511,-86.774,-176.854,11.280,149.475
C04424=1134.179,386.758,-86.813,-176.853,11.282,149.475
C04425=1134.175,387.006,-86.850,-176.852,11.284,149.475
C04426=1134.172,387.253,-86.887,-176.851,11.286,149.475
C04427=1134.167,387.500,-86.924,-176.850,11.288,149.475
C04428=1134.164,387.747,-86.962,-176.849,11.289,149.476
C04429=1134.161,387.994,-87.000,-176.849,11.291,149.476
C04430=1134.157,388.242,-87.037,-176.848,11.292,149.476
C04431=1134.153,388.488,-87.074,-176.847,11.294,149.476
C04432=1134.150,388.701,-87.107,-176.847,11.295,149.477
C04433=1134.147,388.914,-87.139,-176.846,11.297,149.477
C04434=1134.143,389.127,-87.172,-176.845,11.299,149.477
C04435=1134.140,389.340,-87.205,-176.845,11.300,149.477
C04436=1134.137,389.552,-87.236,-176.844,11.302,149.478
C04437=1134.134,389.765,-87.269,-176.844,11.303,149.478
C04438=1134.131,389.978,-87.302,-176.843,11.305,149.478
C04439=1134.127,390.191,-87.334,-176.843,11.306,149.479
C04440=1134.124,390.438,-87.371,-176.842,11.309,149.479
C04441=1134.120,390.684,-87.409,-176.841,11.311,149.479
C04442=1134.117,390.932,-87.446,-176.841,11.313,149.480
C04443=1134.113,391.179,-87.484,-176.840,11.315,149.480
C04444=1134.109,391.425,-87.521,-176.839,11.317,149.480
C04445=1134.105,391.674,-87.559,-176.840,11.318,149.481
C04446=1134.101,391.920,-87.597,-176.839,11.320,149.481
C04447=1134.098,392.168,-87.635,-176.838,11.322,149.482
C04448=1134.094,392.414,-87.672,-176.838,11.325,149.482
C04449=1134.090,392.662,-87.710,-176.837,11.327,149.483
C04450=1134.087,392.909,-87.747,-176.837,11.329,149.483
C04451=1134.083,393.156,-87.786,-176.837,11.331,149.483
C04452=1134.079,393.403,-87.823,-176.837,11.333,149.484
C04453=1134.076,393.651,-87.860,-176.836,11.335,149.484
C04454=1134.072,393.897,-87.898,-176.836,11.337,149.485
C04455=1134.069,394.144,-87.936,-176.835,11.340,149.485
C04456=1134.064,394.391,-87.974,-176.835,11.342,149.486
C04457=1134.061,394.639,-88.011,-176.835,11.344,149.486
C04458=1134.057,394.886,-88.049,-176.835,11.346,149.487
C04459=1134.053,395.132,-88.086,-176.834,11.348,149.487
C04460=1134.049,395.380,-88.125,-176.834,11.351,149.488
C04461=1134.045,395.626,-88.163,-176.834,11.353,149.488
C04462=1134.042,395.874,-88.200,-176.834,11.355,149.489
C04463=1134.038,396.121,-88.237,-176.834,11.358,149.490
C04464=1134.034,396.369,-88.276,-176.833,11.360,149.490
C04465=1134.030,396.615,-88.314,-176.833,11.363,149.491
C04466=1134.027,396.862,-88.351,-176.834,11.364,149.491
C04467=1134.023,397.110,-88.388,-176.834,11.367,149.492
C04468=1134.020,397.357,-88.426,-176.834,11.370,149.493
C04469=1134.015,397.604,-88.464,-176.834,11.372,149.493
C04470=1134.012,397.851,-88.502,-176.834,11.375,149.494
C04471=1134.008,398.098,-88.540,-176.833,11.377,149.495
C04472=1134.005,398.345,-88.578,-176.833,11.380,149.495
C04473=1134.000,398.592,-88.615,-176.833,11.382,149.496
C04474=1133.997,398.840,-88.653,-176.833,11.385,149.496
C04475=1133.993,399.086,-88.691,-176.834,11.388,149.497
C04476=1133.989,399.334,-88.729,-176.833,11.390,149.498
C04477=1133.986,399.580,-88.767,-176.834,11.392,149.499
C04478=1133.982,399.828,-88.805,-176.834,11.395,149.499
C04479=1133.979,400.074,-88.842,-176.835,11.398,149.500
C04480=1133.975,400.322,-88.881,-176.835,11.400,149.501
C04481=1133.971,400.569,-88.918,-176.835,11.403,149.502
C04482=1133.967,400.816,-88.956,-176.835,11.406,149.503
C04483=1133.964,401.063,-88.994,-176.835,11.409,149.503
C04484=1133.960,401.310,-89.032,-176.836,11.412,149.504
C04485=1133.956,401.558,-89.070,-176.836,11.415,149.505
C04486=1133.953,401.804,-89.107,-176.836,11.417,149.506
C04487=1133.949,402.052,-89.146,-176.836,11.420,149.507
C04488=1133.946,402.264,-89.178,-176.837,11.423,149.507
C04489=1133.943,402.476,-89.211,-176.837,11.425,149.508
C04490=1133.939,402.690,-89.243,-176.838,11.428,149.509
C04491=1133.936,402.902,-89.275,-176.838,11.431,149.510
C04492=1133.933,403.115,-89.308,-176.838,11.434,149.510
C04493=1133.930,403.328,-89.341,-176.839,11.435,149.511
C04494=1133.926,403.540,-89.373,-176.839,11.438,149.512
C04495=1133.923,403.753,-89.406,-176.839,11.441,149.513
C04496=1133.919,404.000,-89.444,-176.840,11.444,149.514
C04497=1133.916,404.247,-89.482,-176.841,11.447,149.515
C04498=1133.912,404.494,-89.520,-176.841,11.451,149.516
C04499=1133.908,404.741,-89.558,-176.842,11.454,149.517
C04500=1133.905,404.988,-89.596,-176.842,11.457,149.517
C04501=1133.901,405.235,-89.634,-176.843,11.460,149.518
C04502=1133.898,405.482,-89.672,-176.844,11.463,149.519
C04503=1133.894,405.729,-89.710,-176.844,11.466,149.520
C04504=1133.890,405.977,-89.748,-176.845,11.469,149.521
C04505=1133.886,406.223,-89.786,-176.846,11.473,149.523
C04506=1133.883,406.470,-89.824,-176.847,11.476,149.524
C04507=1133.878,406.718,-89.861,-176.848,11.479,149.525
C04508=1133.875,406.965,-89.899,-176.849,11.483,149.526
C04509=1133.872,407.212,-89.937,-176.849,11.486,149.527
C04510=1133.867,407.459,-89.975,-176.850,11.489,149.528
C04511=1133.864,407.707,-90.013,-176.851,11.494,149.529
C04512=1133.860,407.953,-90.051,-176.852,11.497,149.530
C04513=1133.856,408.201,-90.089,-176.852,11.501,149.531
C04514=1133.852,408.447,-90.127,-176.853,11.504,149.533
C04515=1133.849,408.695,-90.165,-176.855,11.508,149.534
C04516=1133.845,408.942,-90.203,-176.856,11.511,149.535
C04517=1133.842,409.189,-90.241,-176.857,11.515,149.536
C04518=1133.838,409.436,-90.279,-176.858,11.518,149.537
C04519=1133.834,409.682,-90.318,-176.858,11.523,149.539
C04520=1133.831,409.930,-90.356,-176.859,11.526,149.540
C04521=1133.827,410.176,-90.393,-176.861,11.530,149.541
C04522=1133.823,410.424,-90.432,-176.862,11.534,149.542
C04523=1133.819,410.670,-90.469,-176.863,11.537,149.544
C04524=1133.816,410.917,-90.507,-176.864,11.541,149.545
C04525=1133.812,411.165,-90.546,-176.865,11.546,149.546
C04526=1133.809,411.412,-90.583,-176.866,11.549,149.548
C04527=1133.805,411.659,-90.622,-176.868,11.553,149.549
C04528=1133.801,411.906,-90.659,-176.869,11.557,149.550
C04529=1133.798,412.153,-90.697,-176.870,11.562,149.552
C04530=1133.794,412.401,-90.736,-176.872,11.565,149.553
C04531=1133.790,412.647,-90.774,-176.873,11.569,149.554
C04532=1133.787,412.894,-90.811,-176.875,11.573,149.556
C04533=1133.782,413.141,-90.850,-176.876,11.578,149.557
C04534=1133.779,413.389,-90.888,-176.877,11.582,149.559
C04535=1133.775,413.636,-90.926,-176.878,11.586,149.560
C04536=1133.771,413.883,-90.964,-176.880,11.590,149.562
C04537=1133.768,414.130,-91.002,-176.881,11.595,149.563
C04538=1133.764,414.376,-91.041,-176.883,11.599,149.565
C04539=1133.761,414.623,-91.078,-176.884,11.603,149.566
C04540=1133.760,414.871,-91.116,-176.886,11.608,149.568
C04541=1133.758,415.118,-91.154,-176.888,11.612,149.569
C04542=1133.757,415.365,-91.191,-176.889,11.616,149.571
C04543=1133.756,415.612,-91.229,-176.891,11.620,149.572
C04544=1133.757,415.825,-91.262,-176.893,11.624,149.574
C04545=1133.757,416.037,-91.294,-176.894,11.628,149.575
C04546=1133.759,416.250,-91.326,-176.896,11.632,149.576
C04547=1133.760,416.462,-91.358,-176.897,11.636,149.578
C04548=1133.762,416.675,-91.390,-176.899,11.640,149.579
C04549=1133.765,416.888,-91.422,-176.900,11.644,149.581
C04550=1133.767,417.100,-91.453,-176.902,11.648,149.582
C04551=1133.771,417.312,-91.485,-176.903,11.652,149.583
C04552=1133.352,417.312,-91.548,-176.896,11.656,149.583
C04553=1133.349,417.100,-91.517,-176.895,11.652,149.581
C04554=1133.345,416.887,-91.484,-176.893,11.648,149.580
C04555=1133.343,416.675,-91.453,-176.892,11.644,149.579
C04556=1133.341,416.462,-91.421,-176.890,11.640,149.577
C04557=1133.340,416.250,-91.389,-176.888,11.636,149.576
C04558=1133.338,416.037,-91.357,-176.887,11.632,149.574
C04559=1133.337,415.824,-91.324,-176.885,11.628,149.573
C04560=1133.337,415.612,-91.292,-176.884,11.624,149.572
C04561=1133.338,415.365,-91.254,-176.882,11.620,149.570
C04562=1133.338,415.118,-91.216,-176.881,11.616,149.569
C04563=1133.340,414.870,-91.178,-176.879,11.611,149.567
C04564=1133.342,414.624,-91.140,-176.877,11.607,149.565
C04565=1133.345,414.377,-91.103,-176.877,11.603,149.564
C04566=1133.349,414.129,-91.064,-176.875,11.598,149.562
C04567=1133.352,413.882,-91.026,-176.873,11.594,149.561
C04568=1133.356,413.636,-90.989,-176.872,11.589,149.559
C04569=1133.360,413.388,-90.950,-176.871,11.586,149.558
C04570=1133.363,413.141,-90.912,-176.869,11.582,149.557
C04571=1133.367,412.894,-90.874,-176.868,11.577,149.555
C04572=1133.370,412.647,-90.835,-176.867,11.573,149.554
C04573=1133.374,412.401,-90.798,-176.865,11.569,149.553
C04574=1133.378,412.153,-90.759,-176.864,11.565,149.551
C04575=1133.382,411.906,-90.722,-176.863,11.561,149.550
C04576=1133.385,411.659,-90.684,-176.862,11.557,149.548
C04577=1133.389,411.412,-90.645,-176.860,11.553,149.547
C04578=1133.393,411.165,-90.607,-176.860,11.549,149.546
C04579=1133.396,410.917,-90.569,-176.858,11.545,149.544
C04580=1133.400,410.671,-90.531,-176.857,11.541,149.543
C04581=1133.403,410.424,-90.493,-176.856,11.537,149.542
C04582=1133.408,410.177,-90.455,-176.855,11.533,149.541
C04583=1133.411,409.929,-90.417,-176.854,11.530,149.539
C04584=1133.415,409.682,-90.379,-176.853,11.526,149.538
C04585=1133.419,409.435,-90.341,-176.852,11.522,149.537
C04586=1133.422,409.188,-90.303,-176.851,11.518,149.536
C04587=1133.427,408.941,-90.265,-176.850,11.515,149.534
C04588=1133.430,408.694,-90.227,-176.849,11.511,149.533
C04589=1133.434,408.447,-90.190,-176.848,11.507,149.532
C04590=1133.437,408.200,-90.150,-176.847,11.504,149.531
C04591=1133.440,407.953,-90.112,-176.847,11.500,149.530
C04592=1133.444,407.706,-90.075,-176.846,11.496,149.529
C04593=1133.448,407.459,-90.036,-176.845,11.493,149.527
C04594=1133.452,407.212,-89.999,-176.844,11.490,149.526
C04595=1133.455,406.965,-89.961,-176.843,11.486,149.525
C04596=1133.460,406.718,-89.923,-176.842,11.483,149.524
C04597=1133.463,406.471,-89.885,-176.842,11.480,149.523
C04598=1133.466,406.224,-89.847,-176.841,11.476,149.522
C04599=1133.470,405.977,-89.809,-176.841,11.472,149.521
C04600=1133.474,405.729,-89.771,-176.840,11.469,149.520
C04601=1133.477,405.483,-89.733,-176.839,11.466,149.519
C04602=1133.481,405.235,-89.695,-176.839,11.463,149.518
C04603=1133.485,404.989,-89.657,-176.838,11.460,149.517
C04604=1133.489,404.741,-89.620,-176.837,11.456,149.516
C04605=1133.493,404.494,-89.582,-176.836,11.453,149.515
C04606=1133.496,404.247,-89.544,-176.836,11.450,149.514
C04607=1133.500,403.999,-89.506,-176.835,11.447,149.513
C04608=1133.504,403.753,-89.467,-176.836,11.443,149.512
C04609=1133.508,403.540,-89.435,-176.835,11.441,149.512
C04610=1133.510,403.327,-89.403,-176.835,11.438,149.511
C04611=1133.513,403.115,-89.370,-176.834,11.435,149.510
C04612=1133.516,402.902,-89.337,-176.834,11.433,149.509
C04613=1133.519,402.690,-89.304,-176.833,11.431,149.508
C04614=1133.523,402.477,-89.272,-176.833,11.428,149.508
C04615=1133.526,402.264,-89.239,-176.833,11.425,149.507
C04616=1133.529,402.052,-89.206,-176.833,11.422,149.506
C04617=1133.533,401.805,-89.168,-176.832,11.420,149.505
C04618=1133.536,401.558,-89.131,-176.832,11.417,149.504
C04619=1133.540,401.311,-89.092,-176.832,11.414,149.504
C04620=1133.544,401.063,-89.055,-176.831,11.411,149.503
C04621=1133.548,400.816,-89.017,-176.832,11.408,149.502
C04622=1133.552,400.569,-88.979,-176.831,11.406,149.501
C04623=1133.555,400.322,-88.941,-176.831,11.403,149.501
C04624=1133.559,400.075,-88.904,-176.831,11.400,149.500
C04625=1133.562,399.828,-88.866,-176.831,11.397,149.499
C04626=1133.567,399.581,-88.828,-176.831,11.395,149.498
C04627=1133.570,399.334,-88.790,-176.830,11.392,149.498
C04628=1133.573,399.087,-88.752,-176.830,11.389,149.497
C04629=1133.578,398.839,-88.714,-176.831,11.387,149.496
C04630=1133.581,398.592,-88.676,-176.830,11.384,149.495
C04631=1133.585,398.345,-88.639,-176.830,11.382,149.495
C04632=1133.588,398.098,-88.601,-176.830,11.379,149.494
C04633=1133.593,397.851,-88.563,-176.830,11.377,149.494
C04634=1133.596,397.604,-88.525,-176.830,11.374,149.493
C04635=1133.600,397.357,-88.487,-176.830,11.372,149.492
C04636=1133.603,397.109,-88.450,-176.830,11.369,149.492
C04637=1133.608,396.863,-88.412,-176.830,11.367,149.491
C04638=1133.611,396.615,-88.374,-176.831,11.364,149.490
C04639=1133.615,396.369,-88.336,-176.831,11.362,149.490
C04640=1133.618,396.121,-88.298,-176.831,11.359,149.489
C04641=1133.622,395.875,-88.260,-176.831,11.357,149.489
C04642=1133.626,395.627,-88.223,-176.831,11.354,149.488
C04643=1133.630,395.380,-88.185,-176.832,11.352,149.488
C04644=1133.633,395.133,-88.147,-176.832,11.350,149.487
C04645=1133.637,394.886,-88.109,-176.832,11.347,149.487
C04646=1133.641,394.639,-88.072,-176.832,11.346,149.486
C04647=1133.645,394.392,-88.034,-176.832,11.343,149.485
C04648=1133.648,394.145,-87.997,-176.833,11.341,149.485
C04649=1133.652,393.898,-87.959,-176.833,11.339,149.485
C04650=1133.656,393.651,-87.921,-176.834,11.337,149.484
C04651=1133.660,393.403,-87.884,-176.834,11.335,149.484
C04652=1133.663,393.156,-87.846,-176.834,11.332,149.483
C04653=1133.667,392.909,-87.808,-176.835,11.330,149.483
C04654=1133.670,392.663,-87.770,-176.835,11.328,149.482
C04655=1133.675,392.414,-87.733,-176.836,11.326,149.482
C04656=1133.678,392.168,-87.695,-176.836,11.324,149.481
C04657=1133.682,391.920,-87.657,-176.837,11.322,149.481
C04658=1133.685,391.674,-87.620,-176.837,11.320,149.481
C04659=1133.689,391.426,-87.582,-176.837,11.318,149.480
C04660=1133.693,391.179,-87.545,-176.838,11.316,149.480
C04661=1133.697,390.932,-87.506,-176.839,11.314,149.479
C04662=1133.701,390.685,-87.469,-176.840,11.312,149.479
C04663=1133.704,390.438,-87.432,-176.840,11.310,149.479
C04664=1133.708,390.191,-87.394,-176.840,11.308,149.478
C04665=1133.711,389.978,-87.361,-176.841,11.307,149.478
C04666=1133.714,389.765,-87.329,-176.842,11.305,149.478
C04667=1133.717,389.553,-87.297,-176.842,11.304,149.478
C04668=1133.720,389.340,-87.264,-176.843,11.301,149.477
C04669=1133.724,389.127,-87.232,-176.843,11.300,149.477
C04670=1133.727,388.914,-87.200,-176.844,11.299,149.477
C04671=1133.731,388.702,-87.167,-176.845,11.297,149.477
C04672=1133.733,388.489,-87.135,-176.845,11.296,149.476
C04673=1133.737,388.242,-87.098,-176.846,11.294,149.476
C04674=1133.741,387.995,-87.059,-176.847,11.292,149.476
C04675=1133.745,387.747,-87.022,-176.848,11.290,149.476
C04676=1133.748,387.500,-86.985,-176.849,11.288,149.475
C04677=1133.752,387.254,-86.947,-176.850,11.286,149.475
C04678=1133.756,387.006,-86.910,-176.850,11.285,149.475
C04679=1133.759,386.759,-86.872,-176.851,11.283,149.475
C04680=1133.763,386.512,-86.835,-176.852,11.282,149.474
C04681=1133.766,386.265,-86.797,-176.853,11.280,149.474
C04682=1133.770,386.018,-86.760,-176.854,11.278,149.474
C04683=1133.774,385.770,-86.722,-176.855,11.276,149.474
C04684=1133.778,385.523,-86.684,-176.856,11.275,149.474
C04685=1133.782,385.276,-86.648,-176.856,11.273,149.473
C04686=1133.786,385.029,-86.610,-176.858,11.272,149.473
C04687=1133.789,384.782,-86.572,-176.859,11.270,149.473
C04688=1133.793,384.534,-86.535,-176.860,11.268,149.473
C04689=1133.797,384.288,-86.497,-176.861,11.267,149.473
C04690=1133.801,384.041,-86.460,-176.862,11.265,149.473
C04691=1133.804,383.793,-86.422,-176.863,11.264,149.473
C04692=1133.808,383.546,-86.386,-176.864,11.263,149.473
C04693=1133.811,383.299,-86.348,-176.866,11.261,149.473
C04694=1133.815,383.052,-86.311,-176.868,11.259,149.473
C04695=1133.819,382.805,-86.273,-176.871,11.256,149.473
C04696=1133.823,382.557,-86.236,-176.873,11.254,149.473
C04697=1133.827,382.310,-86.198,-176.876,11.252,149.473
C04698=1133.831,382.062,-86.161,-176.879,11.249,149.473
C04699=1133.834,381.816,-86.123,-176.881,11.247,149.473
C04700=1133.838,381.569,-86.086,-176.884,11.244,149.473
C04701=1133.842,381.321,-86.048,-176.886,11.242,149.473
C04702=1133.846,381.074,-86.011,-176.889,11.240,149.473
C04703=1133.849,380.828,-85.974,-176.892,11.237,149.473
C04704=1133.853,380.580,-85.937,-176.894,11.235,149.473
C04705=1133.857,380.333,-85.900,-176.897,11.233,149.473
C04706=1133.861,380.086,-85.862,-176.899,11.231,149.473
C04707=1133.864,379.838,-85.825,-176.902,11.229,149.474
C04708=1133.868,379.591,-85.789,-176.905,11.226,149.474
C04709=1133.872,379.345,-85.751,-176.907,11.224,149.474
C04710=1133.875,379.097,-85.714,-176.910,11.222,149.474
C04711=1133.879,378.850,-85.677,-176.912,11.220,149.474
C04712=1133.883,378.603,-85.639,-176.915,11.217,149.474
C04713=1133.886,378.355,-85.602,-176.918,11.215,149.474
C04714=1133.890,378.108,-85.565,-176.921,11.212,149.474
C04715=1133.894,377.861,-85.528,-176.924,11.211,149.474
C04716=1133.898,377.614,-85.491,-176.926,11.208,149.474
C04717=1133.902,377.366,-85.454,-176.929,11.206,149.475
C04718=1133.906,377.119,-85.417,-176.932,11.203,149.475
C04719=1133.910,376.872,-85.380,-176.935,11.201,149.475
C04720=1133.912,376.625,-85.343,-176.938,11.199,149.475
C04721=1133.916,376.412,-85.311,-176.940,11.197,149.475
C04722=1133.920,376.199,-85.279,-176.943,11.195,149.475
C04723=1133.923,375.986,-85.248,-176.945,11.193,149.475
C04724=1133.927,375.774,-85.215,-176.947,11.191,149.475
C04725=1133.929,375.561,-85.183,-176.950,11.189,149.476
C04726=1133.933,375.348,-85.151,-176.952,11.187,149.476
C04727=1133.936,375.135,-85.120,-176.955,11.185,149.476
C04728=1133.940,374.922,-85.088,-176.957,11.183,149.476
C04729=1133.944,374.675,-85.051,-176.960,11.181,149.476
C04730=1133.946,374.428,-85.014,-176.963,11.179,149.476
C04731=1133.950,374.181,-84.977,-176.966,11.176,149.476
C04732=1133.954,373.933,-84.940,-176.969,11.175,149.477
C04733=1133.958,373.686,-84.904,-176.971,11.172,149.477
C04734=1133.961,373.439,-84.867,-176.974,11.170,149.477
C04735=1133.965,373.192,-84.830,-176.977,11.168,149.477
C04736=1133.969,372.944,-84.793,-176.981,11.165,149.477
C04737=1133.974,372.697,-84.756,-176.983,11.163,149.477
C04738=1133.977,372.450,-84.720,-176.986,11.161,149.478
C04739=1133.980,372.202,-84.683,-176.989,11.159,149.478
C04740=1133.984,371.955,-84.646,-176.992,11.157,149.478
C04741=1133.988,371.708,-84.610,-176.996,11.154,149.478
C04742=1133.992,371.461,-84.573,-176.998,11.152,149.478
C04743=1133.996,371.213,-84.537,-177.001,11.150,149.479
C04744=1134.000,370.966,-84.500,-177.004,11.147,149.479
C04745=1134.003,370.719,-84.463,-177.007,11.146,149.479
C04746=1134.007,370.471,-84.426,-177.010,11.143,149.479
C04747=1134.011,370.224,-84.390,-177.014,11.141,149.479
C04748=1134.015,369.977,-84.353,-177.017,11.138,149.480
C04749=1134.019,369.730,-84.316,-177.020,11.136,149.480
C04750=1134.022,369.483,-84.281,-177.023,11.134,149.480
C04751=1134.027,369.235,-84.244,-177.026,11.131,149.480
C04752=1134.030,368.987,-84.207,-177.029,11.130,149.481
C04753=1134.033,368.741,-84.170,-177.032,11.127,149.481
C04754=1134.037,368.493,-84.134,-177.036,11.125,149.481
C04755=1134.042,368.246,-84.097,-177.039,11.122,149.481
C04756=1134.045,367.999,-84.061,-177.041,11.121,149.481
C04757=1134.049,367.752,-84.024,-177.045,11.118,149.482
C04758=1134.053,367.504,-83.989,-177.048,11.116,149.482
C04759=1134.057,367.257,-83.952,-177.051,11.113,149.482
C04760=1134.060,367.010,-83.916,-177.055,11.111,149.482
C04761=1134.065,366.762,-83.880,-177.057,11.109,149.482
C04762=1134.068,366.515,-83.843,-177.061,11.107,149.483
C04763=1134.072,366.267,-83.806,-177.064,11.104,149.483
C04764=1134.076,366.020,-83.770,-177.067,11.102,149.483
C04765=1134.079,365.773,-83.734,-177.071,11.099,149.483
C04766=1134.084,365.525,-83.697,-177.073,11.097,149.484
C04767=1134.087,365.278,-83.661,-177.077,11.095,149.484
C04768=1134.091,365.031,-83.624,-177.080,11.093,149.484
C04769=1134.095,364.783,-83.589,-177.084,11.090,149.484
C04770=1134.098,364.536,-83.553,-177.087,11.088,149.485
C04771=1134.103,364.289,-83.516,-177.090,11.085,149.485
C04772=1134.106,364.042,-83.480,-177.093,11.083,149.485
C04773=1134.110,363.794,-83.444,-177.097,11.080,149.485
C04774=1134.114,363.547,-83.408,-177.100,11.078,149.485
C04775=1134.118,363.299,-83.372,-177.103,11.076,149.486
C04776=1134.122,363.052,-83.335,-177.106,11.074,149.486
C04777=1134.125,362.839,-83.305,-177.110,11.072,149.486
C04778=1134.128,362.626,-83.274,-177.112,11.070,149.486
C04779=1134.131,362.413,-83.243,-177.115,11.067,149.487
C04780=1134.135,362.200,-83.211,-177.118,11.066,149.487
C04781=1134.139,361.987,-83.181,-177.121,11.064,149.487
C04782=1134.142,361.774,-83.149,-177.124,11.061,149.487
C04783=1134.145,361.562,-83.118,-177.127,11.060,149.488
C04784=1134.148,361.348,-83.087,-177.130,11.057,149.488
C04785=1134.152,361.101,-83.052,-177.133,11.055,149.488
C04786=1134.156,360.854,-83.015,-177.137,11.052,149.488
C04787=1134.159,360.606,-82.979,-177.140,11.050,149.489
C04788=1134.163,360.359,-82.944,-177.144,11.048,149.489
C04789=1134.167,360.111,-82.907,-177.147,11.045,149.489
C04790=1134.171,359.864,-82.872,-177.150,11.043,149.489
C04791=1134.174,359.616,-82.836,-177.154,11.041,149.490
C04792=1134.178,359.369,-82.800,-177.157,11.038,149.490
C04793=1134.183,359.121,-82.764,-177.161,11.036,149.490
C04794=1134.186,358.875,-82.728,-177.164,11.033,149.490
C04795=1134.190,358.627,-82.693,-177.168,11.030,149.491
C04796=1134.194,358.380,-82.657,-177.171,11.028,149.491
C04797=1134.198,358.132,-82.621,-177.175,11.025,149.491
C04798=1134.202,357.885,-82.586,-177.179,11.023,149.492
C04799=1134.206,357.637,-82.550,-177.182,11.021,149.492
C04800=1134.209,357.390,-82.515,-177.185,11.018,149.492
C04801=1134.213,357.143,-82.478,-177.189,11.016,149.492
C04802=1134.218,356.896,-82.442,-177.193,11.013,149.493
C04803=1134.221,356.648,-82.407,-177.196,11.010,149.493
C04804=1134.225,356.401,-82.371,-177.199,11.008,149.493
C04805=1134.229,356.153,-82.336,-177.203,11.006,149.493
C04806=1134.232,355.906,-82.300,-177.206,11.003,149.494
C04807=1134.236,355.658,-82.265,-177.210,11.000,149.494
C04808=1134.240,355.411,-82.229,-177.214,10.998,149.494
C04809=1134.245,355.164,-82.193,-177.217,10.996,149.495
C04810=1134.248,354.916,-82.158,-177.221,10.993,149.495
C04811=1134.252,354.669,-82.122,-177.225,10.990,149.495
C04812=1134.256,354.420,-82.087,-177.228,10.988,149.495
C04813=1134.259,354.173,-82.052,-177.232,10.985,149.496
C04814=1134.264,353.926,-82.017,-177.236,10.982,149.496
C04815=1134.267,353.679,-81.981,-177.239,10.980,149.496
C04816=1134.271,353.431,-81.946,-177.243,10.977,149.496
C04817=1134.275,353.184,-81.910,-177.247,10.974,149.497
C04818=1134.279,352.937,-81.875,-177.250,10.972,149.497
C04819=1134.283,352.689,-81.840,-177.254,10.970,149.497
C04820=1134.287,352.441,-81.805,-177.258,10.967,149.498
C04821=1134.290,352.194,-81.769,-177.261,10.964,149.498
C04822=1134.295,351.947,-81.734,-177.265,10.961,149.498
C04823=1134.299,351.699,-81.699,-177.268,10.958,149.498
C04824=1134.302,351.451,-81.663,-177.272,10.956,149.499
C04825=1134.306,351.204,-81.628,-177.276,10.953,149.499
C04826=1134.310,350.956,-81.593,-177.279,10.951,149.499
C04827=1134.314,350.709,-81.558,-177.284,10.948,149.499
C04828=1134.318,350.461,-81.522,-177.287,10.945,149.500
C04829=1134.322,350.214,-81.488,-177.291,10.942,149.500
C04830=1134.326,349.966,-81.452,-177.295,10.940,149.500
C04831=1134.330,349.719,-81.417,-177.299,10.937,149.500
C04832=1134.334,349.471,-81.382,-177.302,10.934,149.501
C04833=1134.337,349.259,-81.352,-177.305,10.932,149.501
C04834=1134.340,349.045,-81.322,-177.308,10.930,149.501
C04835=1134.344,348.832,-81.291,-177.311,10.927,149.501
C04836=1134.348,348.619,-81.262,-177.314,10.926,149.501
C04837=1134.350,348.406,-81.232,-177.316,10.923,149.502
C04838=1134.354,348.193,-81.201,-177.319,10.921,149.502
C04839=1134.357,347.979,-81.171,-177.322,10.919,149.502
C04840=1134.361,347.766,-81.141,-177.325,10.917,149.502
C04841=1134.364,347.519,-81.106,-177.328,10.914,149.502
C04842=1134.368,347.271,-81.071,-177.331,10.912,149.503
C04843=1134.373,347.024,-81.036,-177.335,10.909,149.503
C04844=1134.376,346.776,-81.001,-177.338,10.907,149.503
C04845=1134.381,346.528,-80.967,-177.341,10.904,149.503
C04846=1134.384,346.281,-80.932,-177.345,10.902,149.503
C04847=1134.388,346.033,-80.897,-177.348,10.899,149.504
C04848=1134.392,345.786,-80.862,-177.351,10.897,149.504
C04849=1134.396,345.538,-80.827,-177.354,10.894,149.504
C04850=1134.400,345.291,-80.793,-177.357,10.892,149.504
C04851=1134.404,345.044,-80.758,-177.361,10.889,149.504
C04852=1134.408,344.795,-80.723,-177.364,10.887,149.505
C04853=1134.412,344.548,-80.688,-177.367,10.884,149.505
C04854=1134.415,344.300,-80.654,-177.371,10.882,149.505
C04855=1134.420,344.053,-80.619,-177.374,10.879,149.505
C04856=1134.424,343.805,-80.584,-177.377,10.877,149.505
C04857=1134.428,343.558,-80.550,-177.380,10.875,149.506
C04858=1134.431,343.310,-80.515,-177.383,10.873,149.506
C04859=1134.436,343.063,-80.480,-177.386,10.870,149.506
C04860=1134.440,342.815,-80.445,-177.390,10.868,149.506
C04861=1134.444,342.568,-80.412,-177.393,10.865,149.506
C04862=1134.448,342.320,-80.377,-177.396,10.862,149.507
C04863=1134.451,342.073,-80.343,-177.399,10.860,149.507
C04864=1134.455,341.825,-80.308,-177.402,10.858,149.507
C04865=1134.460,341.578,-80.273,-177.406,10.855,149.507
C04866=1134.463,341.330,-80.239,-177.409,10.853,149.508
C04867=1134.467,341.083,-80.204,-177.412,10.850,149.508
C04868=1134.471,340.835,-80.169,-177.415,10.847,149.508
C04869=1134.475,340.587,-80.135,-177.419,10.845,149.508
C04870=1134.479,340.339,-80.101,-177.422,10.842,149.508
C04871=1134.483,340.092,-80.067,-177.425,10.840,149.509
C04872=1134.487,339.844,-80.032,-177.429,10.838,149.509
C04873=1134.491,339.597,-79.998,-177.432,10.835,149.509
C04874=1134.495,339.350,-79.964,-177.435,10.832,149.509
C04875=1134.499,339.101,-79.929,-177.438,10.830,149.509
C04876=1134.503,338.854,-79.895,-177.441,10.827,149.510
C04877=1134.507,338.606,-79.860,-177.445,10.825,149.510
C04878=1134.511,338.359,-79.826,-177.448,10.822,149.510
C04879=1134.515,338.111,-79.791,-177.451,10.820,149.510
C04880=1134.519,337.863,-79.758,-177.454,10.817,149.510
C04881=1134.523,337.616,-79.724,-177.458,10.815,149.511
C04882=1134.527,337.368,-79.689,-177.461,10.812,149.511
C04883=1134.531,337.121,-79.656,-177.464,10.810,149.511
C04884=1134.535,336.873,-79.621,-177.467,10.807,149.511
C04885=1134.538,336.626,-79.587,-177.471,10.805,149.511
C04886=1134.543,336.378,-79.552,-177.474,10.802,149.512
C04887=1134.547,336.130,-79.519,-177.477,10.800,149.512
C04888=1134.550,335.883,-79.485,-177.480,10.797,149.512
C04889=1134.554,335.669,-79.455,-177.483,10.795,149.512
C04890=1134.558,335.456,-79.426,-177.486,10.793,149.512
C04891=1134.561,335.242,-79.397,-177.488,10.791,149.513
C04892=1134.565,335.029,-79.368,-177.491,10.788,149.513
C04893=1134.567,334.816,-79.338,-177.494,10.786,149.513
C04894=1134.571,334.603,-79.309,-177.497,10.785,149.513
C04895=1134.575,334.389,-79.279,-177.500,10.782,149.513
C04896=1134.578,334.176,-79.250,-177.502,10.780,149.513
C04897=1134.582,333.928,-79.216,-177.505,10.778,149.514
C04898=1134.586,333.681,-79.182,-177.509,10.775,149.514
C04899=1134.590,333.434,-79.148,-177.512,10.773,149.514
C04900=1134.594,333.185,-79.115,-177.515,10.770,149.514
C04901=1134.598,332.938,-79.080,-177.518,10.767,149.514
C04902=1134.602,332.690,-79.047,-177.521,10.765,149.515
C04903=1134.606,332.442,-79.013,-177.525,10.763,149.515
C04904=1134.609,332.195,-78.979,-177.528,10.760,149.515
C04905=1134.614,331.947,-78.945,-177.531,10.757,149.515
C04906=1134.618,331.700,-78.911,-177.534,10.755,149.515
C04907=1134.622,331.451,-78.878,-177.538,10.752,149.516
C04908=1134.625,331.204,-78.844,-177.541,10.750,149.516
C04909=1134.630,330.956,-78.810,-177.544,10.747,149.516
C04910=1134.634,330.708,-78.776,-177.547,10.745,149.516
C04911=1134.638,330.461,-78.743,-177.551,10.742,149.516
C04912=1134.642,330.214,-78.709,-177.554,10.740,149.517
C04913=1134.646,329.966,-78.676,-177.557,10.737,149.517
C04914=1134.650,329.717,-78.642,-177.560,10.735,149.517
C04915=1134.654,329.470,-78.608,-177.563,10.732,149.517
C04916=1134.658,329.222,-78.575,-177.566,10.729,149.517
C04917=1134.662,328.975,-78.541,-177.570,10.727,149.517
C04918=1134.666,328.728,-78.507,-177.573,10.724,149.518
C04919=1134.669,328.479,-78.474,-177.576,10.722,149.518
C04920=1134.674,328.232,-78.440,-177.579,10.719,149.518
C04921=1134.678,327.984,-78.406,-177.582,10.718,149.518
C04922=1134.682,327.736,-78.373,-177.585,10.715,149.519
C04923=1134.686,327.489,-78.339,-177.589,10.713,149.519
C04924=1134.690,327.241,-78.306,-177.591,10.710,149.519
C04925=1134.694,326.993,-78.273,-177.595,10.707,149.519
C04926=1134.698,326.745,-78.239,-177.598,10.705,149.519
C04927=1134.702,326.498,-78.206,-177.601,10.702,149.519
C04928=1134.706,326.250,-78.172,-177.604,10.700,149.520
C04929=1134.710,326.003,-78.139,-177.608,10.697,149.520
C04930=1134.714,325.754,-78.106,-177.611,10.695,149.520
C04931=1134.718,325.506,-78.073,-177.614,10.692,149.520
C04932=1134.722,325.259,-78.039,-177.617,10.690,149.520
C04933=1134.726,325.012,-78.006,-177.621,10.687,149.521
C04934=1134.730,324.764,-77.972,-177.624,10.684,149.521
C04935=1134.734,324.516,-77.939,-177.627,10.682,149.521
C04936=1134.738,324.268,-77.906,-177.630,10.680,149.521
C04937=1134.742,324.021,-77.873,-177.633,10.677,149.521
C04938=1134.746,323.772,-77.839,-177.636,10.674,149.522
C04939=1134.750,323.525,-77.806,-177.640,10.672,149.522
C04940=1134.754,323.277,-77.773,-177.643,10.669,149.522
C04941=1134.758,323.029,-77.740,-177.646,10.667,149.522
C04942=1134.762,322.781,-77.707,-177.649,10.664,149.522
C04943=1134.766,322.534,-77.674,-177.652,10.661,149.522
C04944=1134.771,322.286,-77.641,-177.656,10.659,149.523
C04945=1134.773,322.072,-77.611,-177.658,10.657,149.523
C04946=1134.777,321.859,-77.583,-177.661,10.655,149.523
C04947=1134.781,321.646,-77.554,-177.663,10.653,149.523
C04948=1134.785,321.432,-77.526,-177.666,10.651,149.523
C04949=1134.787,321.219,-77.498,-177.669,10.648,149.523
C04950=1134.791,321.006,-77.469,-177.672,10.647,149.524
C04951=1134.795,320.792,-77.441,-177.675,10.644,149.524
C04952=1134.798,320.578,-77.413,-177.677,10.642,149.524
C04953=1134.802,320.330,-77.379,-177.680,10.639,149.524
C04954=1134.806,320.082,-77.346,-177.684,10.637,149.524
C04955=1134.810,319.835,-77.313,-177.687,10.634,149.525
C04956=1134.814,319.587,-77.280,-177.690,10.632,149.525
C04957=1134.818,319.340,-77.247,-177.693,10.629,149.525
C04958=1134.822,319.091,-77.215,-177.696,10.626,149.525
C04959=1134.826,318.843,-77.182,-177.700,10.624,149.525
C04960=1134.830,318.596,-77.149,-177.703,10.622,149.526
C04961=1134.834,318.348,-77.116,-177.706,10.619,149.526
C04962=1134.838,318.100,-77.084,-177.709,10.616,149.526
C04963=1134.842,317.852,-77.050,-177.712,10.614,149.526
C04964=1134.846,317.605,-77.018,-177.715,10.611,149.526
C04965=1134.850,317.357,-76.985,-177.718,10.609,149.527
C04966=1134.854,317.109,-76.952,-177.721,10.607,149.527
C04967=1134.859,316.861,-76.919,-177.724,10.604,149.527
C04968=1134.862,316.614,-76.887,-177.728,10.602,149.527
C04969=1134.866,316.365,-76.854,-177.731,10.599,149.527
C04970=1134.871,316.118,-76.821,-177.734,10.597,149.527
C04971=1134.874,315.871,-76.789,-177.737,10.594,149.528
C04972=1134.879,315.622,-76.756,-177.740,10.591,149.528
C04973=1134.883,315.375,-76.723,-177.743,10.589,149.528
C04974=1134.887,315.127,-76.691,-177.747,10.587,149.528
C04975=1134.891,314.879,-76.658,-177.750,10.584,149.528
C04976=1134.895,314.631,-76.626,-177.753,10.581,149.529
C04977=1134.899,314.383,-76.593,-177.756,10.579,149.529
C04978=1134.903,314.135,-76.561,-177.759,10.576,149.529
C04979=1134.907,313.887,-76.528,-177.763,10.574,149.529
C04980=1134.911,313.639,-76.496,-177.766,10.571,149.529
C04981=1134.915,313.391,-76.463,-177.769,10.568,149.530
C04982=1134.920,313.144,-76.431,-177.772,10.566,149.530
C04983=1134.924,312.896,-76.398,-177.775,10.563,149.530
C04984=1134.927,312.648,-76.366,-177.778,10.561,149.530
C04985=1134.931,312.401,-76.333,-177.781,10.558,149.530
C04986=1134.936,312.152,-76.300,-177.785,10.556,149.530
C04987=1134.939,311.905,-76.268,-177.787,10.554,149.531
C04988=1134.944,311.656,-76.235,-177.790,10.551,149.531
C04989=1134.948,311.409,-76.204,-177.794,10.549,149.531
C04990=1134.952,311.161,-76.171,-177.797,10.546,149.531
C04991=1134.956,310.913,-76.139,-177.800,10.544,149.531
C04992=1134.960,310.665,-76.107,-177.803,10.541,149.531
C04993=1134.964,310.418,-76.074,-177.806,10.538,149.532
C04994=1134.968,310.169,-76.042,-177.810,10.536,149.532
C04995=1134.973,309.922,-76.010,-177.812,10.533,149.532
C04996=1134.977,309.673,-75.978,-177.816,10.531,149.532
C04997=1134.980,309.426,-75.945,-177.819,10.528,149.532
C04998=1134.985,309.178,-75.913,-177.822,10.525,149.533
C04999=1134.989,308.930,-75.881,-177.825,10.523,149.533
C05000=1134.993,308.682,-75.849,-177.828,10.520,149.533
C05001=1134.997,308.469,-75.821,-177.831,10.519,149.533
C05002=1135.000,308.256,-75.794,-177.834,10.516,149.533
C05003=1135.004,308.042,-75.766,-177.836,10.514,149.533
C05004=1135.007,307.827,-75.738,-177.839,10.512,149.534
C05005=1135.010,307.614,-75.710,-177.842,10.509,149.534
C05006=1135.014,307.400,-75.683,-177.844,10.507,149.534
C05007=1135.017,307.187,-75.655,-177.848,10.505,149.534
C05008=1135.021,306.973,-75.627,-177.850,10.503,149.534
C05009=1135.026,306.726,-75.595,-177.853,10.501,149.535
C05010=1135.029,306.478,-75.564,-177.856,10.498,149.535
C05011=1135.034,306.230,-75.531,-177.859,10.495,149.535
C05012=1135.037,305.982,-75.499,-177.862,10.493,149.535
C05013=1135.042,305.734,-75.468,-177.866,10.490,149.535
C05014=1135.046,305.486,-75.435,-177.869,10.487,149.535
C05015=1135.050,305.238,-75.403,-177.872,10.485,149.536
C05016=1135.054,304.990,-75.372,-177.875,10.482,149.536
C05017=1135.059,304.742,-75.340,-177.878,10.480,149.536
C05018=1135.062,304.494,-75.308,-177.881,10.478,149.536
C05019=1135.067,304.247,-75.276,-177.884,10.475,149.536
C05020=1135.070,303.999,-75.244,-177.887,10.473,149.537
C05021=1135.075,303.750,-75.212,-177.890,10.470,149.537
C05022=1135.079,303.503,-75.180,-177.893,10.468,149.537
C05023=1135.083,303.254,-75.149,-177.896,10.465,149.537
C05024=1135.087,303.006,-75.117,-177.900,10.463,149.537
C05025=1135.092,302.759,-75.085,-177.903,10.460,149.537
C05026=1135.096,302.511,-75.054,-177.906,10.457,149.538
C05027=1135.099,302.263,-75.022,-177.909,10.455,149.538
C05028=1135.104,302.015,-74.990,-177.912,10.452,149.538
C05029=1135.107,301.767,-74.958,-177.915,10.449,149.538
C05030=1135.113,301.519,-74.927,-177.919,10.447,149.538
C05031=1135.116,301.271,-74.895,-177.922,10.445,149.539
C05032=1135.120,301.023,-74.863,-177.925,10.442,149.539
C05033=1135.124,300.776,-74.832,-177.928,10.439,149.539
C05034=1135.128,300.527,-74.801,-177.930,10.437,149.539
C05035=1135.133,300.280,-74.769,-177.934,10.435,149.539
C05036=1135.136,300.031,-74.737,-177.937,10.432,149.539
C05037=1135.141,299.783,-74.705,-177.940,10.430,149.540
C05038=1135.145,299.535,-74.674,-177.943,10.427,149.540
C05039=1135.149,299.287,-74.642,-177.946,10.425,149.540
C05040=1135.153,299.040,-74.611,-177.949,10.422,149.540
C05041=1135.157,298.791,-74.580,-177.953,10.419,149.540
C05042=1135.162,298.544,-74.548,-177.955,10.417,149.540
C05043=1135.166,298.295,-74.517,-177.959,10.414,149.541
C05044=1135.169,298.047,-74.485,-177.962,10.411,149.541
C05045=1135.174,297.800,-74.454,-177.965,10.409,149.541
C05046=1135.178,297.551,-74.423,-177.968,10.406,149.541
C05047=1135.182,297.304,-74.391,-177.971,10.404,149.541
C05048=1135.186,297.055,-74.360,-177.974,10.401,149.542
C05049=1135.190,296.808,-74.329,-177.978,10.399,149.542
C05050=1135.194,296.559,-74.297,-177.980,10.397,149.542
C05051=1135.199,296.312,-74.266,-177.983,10.394,149.542
C05052=1135.203,296.063,-74.235,-177.986,10.391,149.542
C05053=1135.207,295.816,-74.203,-177.990,10.389,149.543
C05054=1135.211,295.567,-74.172,-177.992,10.386,149.543
C05055=1135.215,295.320,-74.141,-177.996,10.384,149.543
C05056=1135.219,295.071,-74.110,-177.999,10.381,149.543
C05057=1135.223,294.857,-74.083,-178.001,10.379,149.543
C05058=1135.227,294.644,-74.056,-178.004,10.377,149.543
C05059=1135.230,294.430,-74.029,-178.007,10.375,149.543
C05060=1135.234,294.217,-74.003,-178.010,10.372,149.544
C05061=1135.238,294.002,-73.975,-178.012,10.370,149.544
C05062=1135.241,293.789,-73.948,-178.015,10.368,149.544
C05063=1135.245,293.575,-73.921,-178.018,10.365,149.544
C05064=1135.248,293.361,-73.895,-178.020,10.364,149.544
C05065=1135.253,293.113,-73.864,-178.023,10.361,149.544
C05066=1135.256,292.866,-73.833,-178.027,10.359,149.545
C05067=1135.260,292.617,-73.802,-178.029,10.356,149.545
C05068=1135.265,292.369,-73.771,-178.032,10.353,149.545
C05069=1135.269,292.121,-73.740,-178.036,10.351,149.545
C05070=1135.273,291.873,-73.708,-178.039,10.348,149.545
C05071=1135.277,291.625,-73.677,-178.042,10.345,149.546
C05072=1135.281,291.377,-73.647,-178.044,10.343,149.546
C05073=1135.286,291.129,-73.616,-178.048,10.341,149.546
C05074=1135.290,290.880,-73.585,-178.051,10.338,149.546
C05075=1135.294,290.633,-73.554,-178.054,10.336,149.546
C05076=1135.298,290.384,-73.523,-178.057,10.333,149.546
C05077=1135.302,290.137,-73.492,-178.060,10.331,149.547
C05078=1135.306,289.889,-73.462,-178.063,10.328,149.547
C05079=1135.310,289.640,-73.431,-178.067,10.326,149.547
C05080=1135.315,289.392,-73.400,-178.069,10.323,149.547
C05081=1135.319,289.145,-73.370,-178.073,10.320,149.547
C05082=1135.323,288.897,-73.338,-178.076,10.318,149.548
C05083=1135.327,288.649,-73.307,-178.079,10.315,149.548
C05084=1135.331,288.401,-73.277,-178.082,10.312,149.548
C05085=1135.335,288.152,-73.246,-178.084,10.310,149.548
C05086=1135.340,287.904,-73.215,-178.088,10.308,149.548
C05087=1135.344,287.657,-73.185,-178.091,10.305,149.548
C05088=1135.348,287.408,-73.154,-178.094,10.303,149.549
C05089=1135.352,287.160,-73.123,-178.097,10.300,149.549
C05090=1135.356,286.912,-73.093,-178.100,10.298,149.549
C05091=1135.360,286.664,-73.062,-178.103,10.295,149.549
C05092=1135.365,286.416,-73.031,-178.106,10.292,149.549
C05093=1135.369,286.168,-73.001,-178.109,10.290,149.549
C05094=1135.373,285.920,-72.971,-178.112,10.287,149.550
C05095=1135.378,285.671,-72.939,-178.116,10.285,149.550
C05096=1135.381,285.423,-72.909,-178.118,10.283,149.550
C05097=1135.386,285.175,-72.879,-178.121,10.280,149.550
C05098=1135.390,284.928,-72.848,-178.124,10.277,149.550
C05099=1135.394,284.679,-72.817,-178.128,10.275,149.551
C05100=1135.398,284.431,-72.787,-178.131,10.272,149.551
C05101=1135.403,284.183,-72.757,-178.134,10.270,149.551
C05102=1135.407,283.935,-72.726,-178.137,10.267,149.551
C05103=1135.411,283.686,-72.696,-178.140,10.264,149.551
C05104=1135.415,283.438,-72.665,-178.143,10.262,149.551
C05105=1135.419,283.191,-72.635,-178.146,10.259,149.552
C05106=1135.424,282.942,-72.605,-178.149,10.257,149.552
C05107=1135.427,282.694,-72.574,-178.152,10.254,149.552
C05108=1135.432,282.446,-72.543,-178.155,10.252,149.552
C05109=1135.436,282.198,-72.514,-178.158,10.249,149.552
C05110=1135.441,281.950,-72.483,-178.161,10.247,149.552
C05111=1135.445,281.702,-72.453,-178.164,10.244,149.553
C05112=1135.449,281.453,-72.422,-178.167,10.242,149.553
C05113=1135.452,281.223,-72.394,-178.171,10.239,149.553
C05114=1135.456,280.992,-72.367,-178.175,10.236,149.553
C05115=1135.460,280.762,-72.338,-178.178,10.234,149.554
C05116=1135.464,280.531,-72.311,-178.181,10.231,149.554
C05117=1135.469,280.300,-72.282,-178.185,10.228,149.554
C05118=1135.472,280.070,-72.255,-178.188,10.225,149.554
C05119=1135.477,279.839,-72.226,-178.191,10.222,149.554
C05120=1135.480,279.609,-72.198,-178.194,10.220,149.555
C05121=1135.484,279.360,-72.168,-178.198,10.217,149.555
C05122=1135.488,279.112,-72.137,-178.201,10.214,149.555
C05123=1135.493,278.864,-72.108,-178.205,10.211,149.555
C05124=1135.496,278.616,-72.078,-178.209,10.208,149.556
C05125=1135.501,278.367,-72.048,-178.212,10.205,149.556
C05126=1135.506,278.119,-72.018,-178.216,10.203,149.556
C05127=1135.509,277.872,-71.988,-178.220,10.199,149.556
C05128=1135.514,277.623,-71.959,-178.223,10.197,149.556
C05129=1135.518,277.375,-71.928,-178.226,10.194,149.557
C05130=1135.522,277.126,-71.898,-178.229,10.191,149.557
C05131=1135.526,276.878,-71.869,-178.233,10.188,149.557
C05132=1135.531,276.630,-71.838,-178.236,10.185,149.557
C05133=1135.535,276.382,-71.808,-178.240,10.182,149.557
C05134=1135.539,276.134,-71.778,-178.243,10.180,149.557
C05135=1135.543,275.886,-71.749,-178.246,10.177,149.558
C05136=1135.547,275.638,-71.719,-178.249,10.174,149.558
C05137=1135.552,275.389,-71.689,-178.253,10.171,149.558
C05138=1135.556,275.141,-71.659,-178.255,10.168,149.558
C05139=1135.560,274.893,-71.630,-178.259,10.166,149.558
C05140=1135.564,274.645,-71.600,-178.262,10.163,149.558
C05141=1135.585,273.441,-71.457,-177.348,8.390,148.873
C05142=1135.588,273.201,-71.428,-177.351,8.386,148.873
C05143=1135.593,272.961,-71.400,-177.354,8.383,148.872
C05144=1135.597,272.720,-71.371,-177.357,8.380,148.872
C05145=1135.602,272.473,-71.342,-177.359,8.377,148.872
C05146=1135.606,272.225,-71.313,-177.362,8.374,148.872
C05147=1135.610,271.976,-71.284,-177.364,8.371,148.872
C05148=1135.615,271.727,-71.255,-177.367,8.367,148.872
C05149=1135.619,271.479,-71.225,-177.370,8.364,148.872
C05150=1135.622,271.231,-71.196,-177.373,8.361,148.872
C05151=1135.627,270.984,-71.167,-177.375,8.358,148.872
C05152=1135.632,270.735,-71.139,-177.379,8.354,148.872
C05153=1135.636,270.486,-71.109,-177.382,8.351,148.872
C05154=1135.640,270.238,-71.080,-177.384,8.348,148.872
C05155=1135.644,269.989,-71.051,-177.387,8.345,148.872
C05156=1135.649,269.742,-71.022,-177.389,8.342,148.872
C05157=1135.653,269.494,-70.993,-177.392,8.338,148.872
C05158=1135.657,269.245,-70.964,-177.395,8.335,148.872
C05159=1135.661,268.997,-70.935,-177.398,8.332,148.872
C05160=1135.665,268.748,-70.905,-177.400,8.329,148.872
C05161=1135.671,268.500,-70.877,-177.403,8.326,148.872
C05162=1135.674,268.252,-70.848,-177.406,8.322,148.872
C05163=1135.678,268.003,-70.819,-177.409,8.319,148.872
C05164=1135.683,267.755,-70.790,-177.412,8.316,148.872
C05165=1135.687,267.508,-70.761,-177.414,8.313,148.872
C05166=1135.691,267.259,-70.733,-177.417,8.310,148.872
C05167=1135.695,267.011,-70.703,-177.420,8.306,148.872
C05168=1135.700,266.762,-70.674,-177.423,8.303,148.872
C05169=1135.705,266.514,-70.645,-177.425,8.300,148.872
C05170=1135.708,266.266,-70.617,-177.428,8.297,148.872
C05171=1135.713,266.017,-70.588,-177.431,8.294,148.872
C05172=1135.718,265.769,-70.559,-177.434,8.291,148.872
C05173=1135.722,265.521,-70.530,-177.437,8.287,148.872
C05174=1135.726,265.272,-70.502,-177.439,8.284,148.872
C05175=1135.731,265.024,-70.473,-177.442,8.281,148.872
C05176=1135.735,264.776,-70.444,-177.445,8.278,148.872
C05177=1135.739,264.527,-70.416,-177.447,8.275,148.872
C05178=1135.743,264.280,-70.387,-177.451,8.272,148.872
C05179=1135.747,264.031,-70.359,-177.454,8.269,148.872
C05180=1135.752,263.782,-70.330,-177.456,8.265,148.872
C05181=1135.756,263.535,-70.301,-177.459,8.262,148.872
C05182=1135.760,263.286,-70.273,-177.462,8.260,148.872
C05183=1135.765,263.037,-70.244,-177.464,8.257,148.872
C05184=1135.770,262.789,-70.216,-177.467,8.253,148.872
C05185=1135.773,262.541,-70.187,-177.470,8.250,148.872
C05186=1135.778,262.292,-70.158,-177.473,8.247,148.872
C05187=1135.782,262.044,-70.130,-177.476,8.244,148.872
C05188=1135.787,261.795,-70.101,-177.478,8.241,148.872
C05189=1135.791,261.523,-70.070,-177.481,8.237,148.872
C05190=1135.796,261.248,-70.038,-177.484,8.234,148.872
C05191=1135.800,260.975,-70.008,-177.488,8.230,148.872
C05192=1135.805,260.702,-69.976,-177.491,8.226,148.872
C05193=1135.810,260.453,-69.947,-177.493,8.223,148.872
C05194=1135.814,260.205,-69.919,-177.496,8.220,148.872
C05195=1135.818,259.957,-69.891,-177.499,8.217,148.872
C05196=1135.823,259.708,-69.862,-177.502,8.214,148.872
C05197=1135.827,259.460,-69.835,-177.504,8.212,148.872
C05198=1135.831,259.211,-69.806,-177.507,8.208,148.872
C05199=1135.836,258.963,-69.778,-177.510,8.205,148.872
C05200=1135.840,258.714,-69.749,-177.513,8.202,148.872
C05201=1135.844,258.466,-69.721,-177.516,8.199,148.872
C05202=1135.849,258.217,-69.693,-177.518,8.195,148.872
C05203=1135.852,257.970,-69.664,-177.521,8.193,148.872
C05204=1135.857,257.722,-69.636,-177.524,8.190,148.872
C05205=1135.861,257.473,-69.607,-177.527,8.187,148.872
C05206=1135.866,257.224,-69.580,-177.530,8.183,148.872
C05207=1135.870,256.975,-69.552,-177.532,8.180,148.872
C05208=1135.875,256.728,-69.524,-177.535,8.177,148.872
C05209=1135.879,256.479,-69.496,-177.538,8.174,148.872
C05210=1135.884,256.231,-69.467,-177.541,8.171,148.872
C05211=1135.887,255.982,-69.439,-177.543,8.168,148.872
C05212=1135.892,255.734,-69.411,-177.546,8.165,148.872
C05213=1135.896,255.485,-69.383,-177.549,8.162,148.872
C05214=1135.901,255.238,-69.355,-177.552,8.158,148.872
C05215=1135.904,254.989,-69.327,-177.555,8.155,148.872
C05216=1135.910,254.740,-69.299,-177.558,8.152,148.873
C05217=1135.914,254.492,-69.271,-177.560,8.149,148.873
C05218=1135.918,254.244,-69.243,-177.563,8.146,148.872
C05219=1135.922,253.996,-69.215,-177.566,8.143,148.873
C05220=1135.927,253.747,-69.187,-177.568,8.140,148.873
C05221=1135.931,253.498,-69.160,-177.571,8.137,148.873
C05222=1135.935,253.250,-69.131,-177.574,8.135,148.873
C05223=1135.939,253.002,-69.104,-177.577,8.132,148.873
C05224=1135.945,252.754,-69.075,-177.580,8.128,148.873
C05225=1135.949,252.505,-69.048,-177.582,8.125,148.873
C05226=1135.953,252.257,-69.020,-177.585,8.122,148.873
C05227=1135.957,252.008,-68.992,-177.588,8.119,148.873
C05228=1135.961,251.760,-68.965,-177.591,8.116,148.873
C05229=1135.966,251.512,-68.937,-177.594,8.113,148.873
C05230=1135.970,251.263,-68.908,-177.596,8.110,148.873
C05231=1135.975,251.014,-68.881,-177.599,8.107,148.873
C05232=1135.979,250.766,-68.853,-177.602,8.104,148.873
C05233=1135.983,250.518,-68.825,-177.604,8.101,148.873
C05234=1135.988,250.269,-68.798,-177.607,8.098,148.873
C05235=1135.991,250.021,-68.770,-177.611,8.094,148.873
C05236=1135.996,249.772,-68.743,-177.613,8.092,148.873
C05237=1136.001,249.524,-68.715,-177.616,8.089,148.873
C05238=1136.005,249.275,-68.687,-177.619,8.086,148.873
C05239=1136.009,249.027,-68.660,-177.621,8.082,148.873
C05240=1136.014,248.779,-68.632,-177.624,8.080,148.873
C05241=1136.018,248.530,-68.604,-177.627,8.077,148.873
C05242=1136.023,248.282,-68.577,-177.630,8.074,148.873
C05243=1136.027,248.034,-68.550,-177.633,8.071,148.874
C05244=1136.031,247.784,-68.522,-177.635,8.068,148.874
C05245=1136.035,247.537,-68.494,-177.638,8.065,148.874
C05246=1136.040,247.288,-68.467,-177.641,8.062,148.874
C05247=1136.044,247.040,-68.439,-177.644,8.059,148.874
C05248=1136.048,246.791,-68.412,-177.647,8.056,148.874
C05249=1136.053,246.543,-68.385,-177.649,8.053,148.874
C05250=1136.057,246.295,-68.357,-177.652,8.049,148.874
C05251=1136.061,246.045,-68.330,-177.655,8.046,148.874
C05252=1136.066,245.797,-68.303,-177.658,8.043,148.874
C05253=1136.070,245.549,-68.275,-177.661,8.041,148.874
C05254=1136.075,245.301,-68.248,-177.664,8.038,148.874
C05255=1136.079,245.051,-68.220,-177.666,8.035,148.874
C05256=1136.083,244.804,-68.193,-177.669,8.032,148.874
C05257=1136.088,244.555,-68.166,-177.672,8.029,148.874
C05258=1136.093,244.307,-68.139,-177.675,8.026,148.874
C05259=1136.097,244.057,-68.111,-177.678,8.023,148.875
C05260=1136.101,243.809,-68.083,-177.680,8.020,148.875
C05261=1136.105,243.561,-68.057,-177.683,8.017,148.874
C05262=1136.110,243.313,-68.030,-177.686,8.014,148.875
C05263=1136.114,243.064,-68.003,-177.688,8.011,148.875
C05264=1136.118,242.815,-67.975,-177.691,8.008,148.875
C05265=1136.123,242.567,-67.948,-177.694,8.005,148.875
C05266=1136.128,242.319,-67.920,-177.697,8.002,148.875
C05267=1136.132,242.070,-67.893,-177.700,7.999,148.875
C05268=1136.136,241.822,-67.867,-177.702,7.997,148.875
C05269=1136.141,241.574,-67.840,-177.705,7.994,148.875
C05270=1136.145,241.324,-67.812,-177.708,7.991,148.875
C05271=1136.149,241.076,-67.785,-177.711,7.988,148.875
C05272=1136.154,240.827,-67.758,-177.714,7.985,148.875
C05273=1136.158,240.579,-67.732,-177.716,7.982,148.875
C05274=1136.163,240.331,-67.705,-177.719,7.979,148.876
C05275=1136.167,240.082,-67.678,-177.722,7.976,148.876
C05276=1136.172,239.834,-67.651,-177.725,7.973,148.876
C05277=1136.175,239.585,-67.624,-177.728,7.970,148.876
C05278=1136.180,239.336,-67.597,-177.730,7.967,148.876
C05279=1136.185,239.088,-67.570,-177.733,7.965,148.876
C05280=1136.189,238.839,-67.543,-177.736,7.962,148.876
C05281=1136.193,238.591,-67.516,-177.739,7.959,148.876
C05282=1136.198,238.343,-67.489,-177.742,7.956,148.876
C05283=1136.203,238.094,-67.462,-177.744,7.953,148.876
C05284=1136.206,237.846,-67.436,-177.747,7.950,148.876
C05285=1136.211,237.597,-67.409,-177.750,7.947,148.876
C05286=1136.216,237.349,-67.381,-177.753,7.944,148.877
C05287=1136.220,237.101,-67.355,-177.756,7.941,148.877
C05288=1136.224,236.851,-67.328,-177.758,7.938,148.877
C05289=1136.229,236.602,-67.301,-177.761,7.935,148.877
C05290=1136.233,236.354,-67.275,-177.764,7.933,148.877
C05291=1136.237,236.106,-67.248,-177.767,7.930,148.877
C05292=1136.242,235.857,-67.221,-177.770,7.927,148.877
C05293=1136.247,235.585,-67.193,-177.773,7.923,148.877
C05294=1136.252,235.314,-67.163,-177.776,7.920,148.877
C05295=1136.256,235.041,-67.134,-177.779,7.917,148.877
C05296=1136.261,234.770,-67.104,-177.782,7.913,148.877
C05297=1136.266,234.521,-67.078,-177.785,7.911,148.877
C05298=1136.270,234.273,-67.051,-177.788,7.908,148.877
C05299=1136.274,234.024,-67.025,-177.790,7.905,148.878
C05300=1136.279,233.775,-66.999,-177.793,7.902,148.878
C05301=1136.283,233.527,-66.972,-177.796,7.899,148.878
C05302=1136.288,233.279,-66.945,-177.799,7.896,148.878
C05303=1136.293,233.029,-66.919,-177.802,7.893,148.878
C05304=1136.297,232.781,-66.892,-177.804,7.891,148.878
C05305=1136.302,232.532,-66.866,-177.807,7.888,148.878
C05306=1136.305,232.284,-66.839,-177.809,7.885,148.878
C05307=1136.309,232.036,-66.813,-177.812,7.882,148.878
C05308=1136.314,231.787,-66.787,-177.816,7.880,148.879
C05309=1136.318,231.539,-66.760,-177.818,7.877,148.879
C05310=1136.323,231.289,-66.734,-177.821,7.874,148.879
C05311=1136.327,231.041,-66.707,-177.824,7.871,148.879
C05312=1136.332,230.792,-66.681,-177.827,7.868,148.879
C05313=1136.336,230.544,-66.655,-177.830,7.865,148.879
C05314=1136.342,230.295,-66.629,-177.832,7.862,148.879
C05315=1136.346,230.047,-66.602,-177.835,7.859,148.879
C05316=1136.350,229.799,-66.576,-177.838,7.857,148.879
C05317=1136.354,229.550,-66.549,-177.841,7.854,148.879
C05318=1136.359,229.301,-66.524,-177.844,7.851,148.879
C05319=1136.363,229.053,-66.496,-177.846,7.848,148.880
C05320=1136.368,228.804,-66.471,-177.849,7.845,148.880
C05321=1136.372,228.555,-66.445,-177.852,7.842,148.880
C05322=1136.376,228.307,-66.418,-177.855,7.839,148.880
C05323=1136.381,228.059,-66.393,-177.858,7.837,148.880
C05324=1136.385,227.810,-66.366,-177.860,7.834,148.880
C05325=1136.390,227.561,-66.340,-177.863,7.832,148.880
C05326=1136.394,227.312,-66.314,-177.866,7.829,148.880
C05327=1136.399,227.064,-66.288,-177.869,7.826,148.880
C05328=1136.403,226.815,-66.261,-177.872,7.823,148.881
C05329=1136.407,226.566,-66.235,-177.874,7.820,148.881
C05330=1136.412,226.318,-66.210,-177.877,7.817,148.881
C05331=1136.416,226.070,-66.184,-177.880,7.814,148.881
C05332=1136.421,225.821,-66.157,-177.883,7.811,148.881
C05333=1136.425,225.572,-66.131,-177.886,7.809,148.881
C05334=1136.430,225.323,-66.106,-177.889,7.806,148.881
C05335=1136.434,225.076,-66.080,-177.891,7.804,148.881
C05336=1136.439,224.827,-66.053,-177.894,7.801,148.882
C05337=1136.443,224.578,-66.027,-177.897,7.798,148.882
C05338=1136.448,224.329,-66.002,-177.900,7.795,148.882
C05339=1136.452,224.080,-65.976,-177.902,7.792,148.882
C05340=1136.457,223.832,-65.951,-177.905,7.789,148.882
C05341=1136.462,223.583,-65.924,-177.908,7.786,148.882
C05342=1136.465,223.335,-65.898,-177.911,7.784,148.882
C05343=1136.470,223.086,-65.872,-177.914,7.781,148.882
C05344=1136.475,222.838,-65.847,-177.917,7.778,148.883
C05345=1136.479,222.589,-65.821,-177.919,7.776,148.883
C05346=1136.483,222.340,-65.795,-177.922,7.773,148.883
C05347=1136.487,222.092,-65.769,-177.925,7.770,148.883
C05348=1136.493,221.843,-65.743,-177.927,7.767,148.883
C05349=1136.497,221.594,-65.718,-177.931,7.764,148.883
C05350=1136.501,221.346,-65.692,-177.934,7.762,148.883
C05351=1136.505,221.097,-65.666,-177.936,7.759,148.883
C05352=1136.510,220.849,-65.641,-177.939,7.756,148.884
C05353=1136.514,220.600,-65.615,-177.941,7.754,148.884
C05354=1136.519,220.351,-65.589,-177.944,7.751,148.884
C05355=1136.524,220.103,-65.564,-177.947,7.748,148.884
C05356=1136.528,219.854,-65.538,-177.950,7.745,148.884
C05357=1136.532,219.605,-65.512,-177.953,7.742,148.884
C05358=1136.537,219.357,-65.487,-177.956,7.740,148.884
C05359=1136.541,219.108,-65.462,-177.959,7.737,148.884
C05360=1136.546,218.859,-65.436,-177.962,7.734,148.885
C05361=1136.550,218.611,-65.411,-177.964,7.732,148.885
C05362=1136.555,218.362,-65.385,-177.967,7.729,148.885
C05363=1136.559,218.113,-65.359,-177.970,7.726,148.885
C05364=1136.564,217.865,-65.334,-177.973,7.723,148.885
C05365=1136.568,217.616,-65.309,-177.975,7.720,148.885
C05366=1136.572,217.367,-65.283,-177.979,7.718,148.886
C05367=1136.577,217.119,-65.258,-177.982,7.715,148.886
C05368=1136.581,216.870,-65.232,-177.984,7.713,148.886
C05369=1136.586,216.622,-65.207,-177.987,7.710,148.886
C05370=1136.591,216.372,-65.182,-177.989,7.707,148.886
C05371=1136.595,216.124,-65.156,-177.993,7.704,148.886
C05372=1136.600,215.876,-65.130,-177.995,7.702,148.886
C05373=1136.604,215.626,-65.105,-177.998,7.699,148.886
C05374=1136.608,215.378,-65.081,-178.000,7.697,148.887
C05375=1136.613,215.130,-65.055,-178.003,7.694,148.887
C05376=1136.617,214.880,-65.030,-178.007,7.691,148.887
C05377=1136.622,214.632,-65.004,-178.009,7.688,148.887
C05378=1136.626,214.383,-64.979,-178.012,7.685,148.887
C05379=1136.631,214.134,-64.954,-178.015,7.682,148.887
C05380=1136.636,213.886,-64.928,-178.018,7.681,148.888
C05381=1136.640,213.638,-64.904,-178.020,7.678,148.888
C05382=1136.644,213.388,-64.878,-178.023,7.675,148.888
C05383=1136.648,213.140,-64.853,-178.026,7.672,148.888
C05384=1136.654,212.891,-64.828,-178.029,7.669,148.888
C05385=1136.658,212.642,-64.802,-178.032,7.667,148.888
C05386=1136.662,212.394,-64.778,-178.034,7.664,148.889
C05387=1136.666,212.145,-64.752,-178.037,7.662,148.889
C05388=1136.672,211.896,-64.728,-178.040,7.659,148.889
C05389=1136.676,211.647,-64.702,-178.043,7.656,148.889
C05390=1136.681,211.399,-64.677,-178.046,7.653,148.889
C05391=1136.684,211.150,-64.652,-178.048,7.651,148.889
C05392=1136.690,210.901,-64.628,-178.052,7.649,148.890
C05393=1136.694,210.653,-64.602,-178.054,7.646,148.890
C05394=1136.698,210.404,-64.578,-178.057,7.643,148.890
C05395=1136.702,210.155,-64.552,-178.060,7.640,148.890
C05396=1136.708,209.907,-64.527,-178.063,7.638,148.890
C05397=1136.712,209.636,-64.500,-178.066,7.635,148.890
C05398=1136.717,209.366,-64.474,-178.069,7.631,148.890
C05399=1136.722,209.095,-64.446,-178.072,7.629,148.891
C05400=1136.727,208.824,-64.419,-178.075,7.626,148.891
C05401=1136.731,208.575,-64.395,-178.078,7.623,148.891
C05402=1136.736,208.327,-64.369,-178.081,7.621,148.891
C05403=1136.741,208.078,-64.344,-178.083,7.619,148.891
C05404=1136.745,207.829,-64.320,-178.086,7.616,148.892
C05405=1136.749,207.580,-64.294,-178.089,7.613,148.892
C05406=1136.755,207.332,-64.270,-178.092,7.610,148.892
C05407=1136.759,207.083,-64.246,-178.094,7.608,148.892
C05408=1136.764,206.834,-64.221,-178.098,7.606,148.892
C05409=1136.768,206.586,-64.196,-178.101,7.603,148.893
C05410=1136.772,206.337,-64.171,-178.103,7.600,148.893
C05411=1136.777,206.088,-64.147,-178.106,7.598,148.893
C05412=1136.782,205.840,-64.122,-178.109,7.595,148.893
C05413=1136.786,205.590,-64.097,-178.112,7.592,148.893
C05414=1136.791,205.342,-64.073,-178.115,7.589,148.893
C05415=1136.795,205.094,-64.048,-178.117,7.588,148.894
C05416=1136.799,204.844,-64.023,-178.120,7.585,148.894
C05417=1136.804,204.596,-63.999,-178.123,7.582,148.894
C05418=1136.809,204.347,-63.974,-178.126,7.579,148.894
C05419=1136.813,204.098,-63.949,-178.128,7.577,148.894
C05420=1136.818,203.849,-63.925,-178.131,7.574,148.894
C05421=1136.823,203.601,-63.901,-178.134,7.572,148.895
C05422=1136.827,203.352,-63.876,-178.137,7.569,148.895
C05423=1136.832,203.103,-63.852,-178.139,7.567,148.895
C05424=1136.836,202.855,-63.827,-178.143,7.564,148.895
C05425=1136.841,202.605,-63.802,-178.146,7.561,148.895
C05426=1136.845,202.357,-63.778,-178.149,7.559,148.896
C05427=1136.849,202.108,-63.754,-178.151,7.557,148.896
C05428=1136.854,201.859,-63.729,-178.154,7.554,148.896
C05429=1136.858,201.610,-63.705,-178.157,7.551,148.896
C05430=1136.863,201.362,-63.681,-178.159,7.549,148.896
C05431=1136.867,201.113,-63.656,-178.162,7.546,148.897
C05432=1136.872,200.864,-63.632,-178.165,7.544,148.897
C05433=1136.877,200.615,-63.607,-178.168,7.541,148.897
C05434=1136.881,200.367,-63.583,-178.171,7.539,148.897
C05435=1136.885,200.118,-63.559,-178.174,7.536,148.897
C05436=1136.890,199.869,-63.534,-178.177,7.533,148.898
C05437=1136.895,199.620,-63.511,-178.179,7.532,148.898
C05438=1136.900,199.371,-63.486,-178.182,7.529,148.898
C05439=1136.904,199.122,-63.462,-178.185,7.526,148.898
C05440=1136.908,198.874,-63.438,-178.188,7.523,148.898
C05441=1136.913,198.626,-63.414,-178.190,7.521,148.899
C05442=1136.918,198.377,-63.389,-178.194,7.519,148.899
C05443=1136.922,198.128,-63.365,-178.197,7.516,148.899
C05444=1136.926,197.879,-63.341,-178.199,7.514,148.899
C05445=1136.931,197.630,-63.316,-178.202,7.511,148.900
C05446=1136.936,197.382,-63.292,-178.205,7.508,148.900
C05447=1136.940,197.132,-63.269,-178.208,7.506,148.900
C05448=1136.945,196.884,-63.245,-178.210,7.503,148.900
